KUKA KRL program: MyProgram_046().src

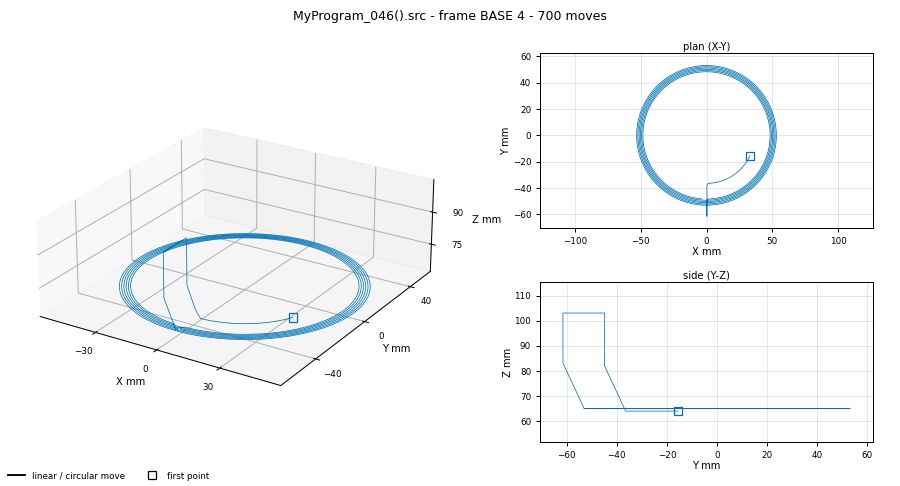
[picture p0: tool path of MyProgram_046().src in frame BASE 4, 700 of 700 moves have a stored position in this frame; points joined in program order, loops and branches not executed]
&ACCESS RVP
&REL 1
&PARAM TEMPLATE = C:\KRC\Roboter\Template\vorgabe
&PARAM EDITMASK = *
DEF MyProgram_046()
; ---- Setting reference (Base) ----
$BASE = BASE_DATA[4]

; --------------------------
; ---- Setting tool (TCP) ----
$TOOL = TOOL_DATA[3]
; --------------------------

$VEL.CP = VEL_APROX_PRINT
Startdeposition()
$VEL.CP = VEL_PRINT
LIN {X 32.9822,Y -15.5864,Z 64,A -32.7373,B 24.8477,C -2.8475,E1 25.1437,E2 -244.1821} C_DIS
LIN {X 32.179,Y -17.1845,Z 64,A -35.4809,B 24.8484,C -2.8403,E1 25.1402,E2 -241.4362} C_DIS
LIN {X 31.292,Y -18.7512,Z 64,A -38.3533,B 24.8494,C -2.8317,E1 25.1362,E2 -238.5581} C_DIS
LIN {X 30.3289,Y -20.2722,Z 64,A -41.1594,B 24.8502,C -2.8242,E1 25.1319,E2 -235.7483} C_DIS
LIN {X 29.3067,Y -21.7235,Z 64,A -44.1232,B 24.8512,C -2.8142,E1 25.127,E2 -232.7751} C_DIS
LIN {X 27.9176,Y -23.4819,Z 64,A -47.6149,B 24.8521,C -2.8055,E1 25.1208,E2 -229.2792} C_DIS
LIN {X 26.4275,Y -25.1472,Z 64,A -51.129,B 24.8531,C -2.7969,E1 25.1142,E2 -225.76} C_DIS
LIN {X 24.8238,Y -26.7316,Z 64,A -54.6334,B 24.8539,C -2.7891,E1 25.1071,E2 -222.2517} C_DIS
LIN {X 23.1454,Y -28.1974,Z 64,A -58.1204,B 24.8547,C -2.7816,E1 25.0997,E2 -218.7605} C_DIS
LIN {X 21.3705,Y -29.5653,Z 64,A -61.4314,B 24.8551,C -2.7774,E1 25.0923,E2 -215.4513} C_DIS
LIN {X 19.9064,Y -30.57,Z 64,A -64.2082,B 24.8557,C -2.7722,E1 25.0858,E2 -212.6714} C_DIS
LIN {X 17.934,Y -31.767,Z 64,A -67.344,B 24.8557,C -2.7725,E1 25.0783,E2 -209.5461} C_DIS
LIN {X 16.1118,Y -32.7286,Z 64,A -71.1277,B 24.857,C -2.7596,E1 25.0689,E2 -205.7422} C_DIS
LIN {X 14.241,Y -33.5852,Z 64,A -74.4803,B 24.8576,C -2.7532,E1 25.0603,E2 -202.3826} C_DIS
LIN {X 12.2935,Y -34.3456,Z 64,A -77.5119,B 24.8577,C -2.7523,E1 25.0524,E2 -199.3554} C_DIS
LIN {X 10.5964,Y -34.9065,Z 64,A -80.3398,B 24.8581,C -2.7487,E1 25.0448,E2 -196.5242} C_DIS
LIN {X 8.8621,Y -35.387,Z 64,A -83.152,B 24.8584,C -2.746,E1 25.0372,E2 -193.71} C_DIS
LIN {X 7.1184,Y -35.7786,Z 64,A -86.157,B 24.8589,C -2.741,E1 25.029,E2 -190.6968} C_DIS
LIN {X 4.917,Y -36.1471,Z 64,A -89.4787,B 24.8589,C -2.741,E1 25.0199,E2 -187.3781} C_DIS
LIN {X 3.1411,Y -36.3441,Z 64,A -92.2456,B 24.859,C -2.7399,E1 25.0122,E2 -184.6106} C_DIS
LIN {X 1.2285,Y -36.4591,Z 64,A -95.4915,B 24.8594,C -2.7358,E1 25.0031,E2 -181.356} C_DIS
LIN {X 1.2285,Y -36.4591,Z 64,A -95.4915,B 24.8594,C -2.7358,E1 25.0031,E2 -181.356} C_DIS
Enddeposition()
LIN {X 0.2612,Y -38.5893,Z 68.5315,A -95.5236,B 24.858,C -2.7494,E1 25.0031,E2 -181.356} C_DIS
LIN {X 0.3711,Y -44.9276,Z 82.1262,A -95.4901,B 24.8595,C -2.7353,E1 25.0031,E2 -181.356} C_DIS
LIN {X 0.3711,Y -44.9276,Z 103.1262,A -95.8409,B 24.8439,C -2.8827,E1 25.0031,E2 -181.356} C_DIS
LIN {X 0.2647,Y -61.4887,Z 103.1262,A -96.1468,B 24.8737,C -2.5936,E1 25.0003,E2 -180.3627} C_DIS
LIN {X 0.2647,Y -61.4887,Z 83.1262,A -95.8133,B 24.887,C -2.4533,E1 25.0003,E2 -180.3627} C_DIS
LIN {X 0.2647,Y -55.1494,Z 69.5315,A -95.8444,B 24.8858,C -2.4664,E1 25.0003,E2 -180.3627} C_DIS
LIN {X 0.2647,Y -53.0363,Z 65,A -95.8563,B 24.8854,C -2.4714,E1 25.0003,E2 -180.3627} C_DIS
Startdeposition()
$VEL.CP = VEL_PRINT
LIN {X -1.9523,Y -53.0044,Z 65,A -98.6503,B 24.8861,C -2.4637,E1 24.9925,E2 -177.5499} C_DIS
LIN {X -4.5507,Y -52.8447,Z 65,A -101.4628,B 24.8861,C -2.4637,E1 24.9846,E2 -174.7363} C_DIS
LIN {X -7.1382,Y -52.5578,Z 65,A -104.2762,B 24.8861,C -2.4641,E1 24.9768,E2 -171.9219} C_DIS
LIN {X -9.7085,Y -52.1442,Z 65,A -107.0908,B 24.886,C -2.4649,E1 24.9691,E2 -169.1066} C_DIS
LIN {X -12.2554,Y -51.605,Z 65,A -109.9063,B 24.8858,C -2.4662,E1 24.9614,E2 -166.2905} C_DIS
LIN {X -14.7728,Y -50.9415,Z 65,A -112.7228,B 24.8857,C -2.4679,E1 24.9538,E2 -163.4736} C_DIS
LIN {X -17.2546,Y -50.1553,Z 65,A -115.5402,B 24.8855,C -2.4699,E1 24.9464,E2 -160.6559} C_DIS
LIN {X -19.6948,Y -49.2482,Z 65,A -118.3587,B 24.8853,C -2.4724,E1 24.939,E2 -157.8374} C_DIS
LIN {X -22.0875,Y -48.2225,Z 65,A -121.178,B 24.885,C -2.4753,E1 24.9318,E2 -155.0181} C_DIS
LIN {X -24.4271,Y -47.0807,Z 65,A -123.9982,B 24.8847,C -2.4786,E1 24.9248,E2 -152.1982} C_DIS
LIN {X -26.7078,Y -45.8254,Z 65,A -126.8195,B 24.8844,C -2.4822,E1 24.9179,E2 -149.3774} C_DIS
LIN {X -28.9242,Y -44.4597,Z 65,A -129.6416,B 24.884,C -2.4863,E1 24.9113,E2 -146.5559} C_DIS
LIN {X -31.0709,Y -42.9869,Z 65,A -132.4651,B 24.8836,C -2.4906,E1 24.9048,E2 -143.7331} C_DIS
LIN {X -33.1427,Y -41.4105,Z 65,A -135.2883,B 24.8831,C -2.4954,E1 24.8986,E2 -140.911} C_DIS
LIN {X -35.1347,Y -39.7344,Z 65,A -138.1128,B 24.8826,C -2.5005,E1 24.8926,E2 -138.0876} C_DIS
LIN {X -37.0421,Y -37.9626,Z 65,A -140.9383,B 24.8821,C -2.5059,E1 24.8869,E2 -135.2634} C_DIS
LIN {X -38.8602,Y -36.0993,Z 65,A -143.7646,B 24.8816,C -2.5117,E1 24.8815,E2 -132.4386} C_DIS
LIN {X -40.5847,Y -34.149,Z 65,A -146.5914,B 24.881,C -2.5178,E1 24.8763,E2 -129.6134} C_DIS
LIN {X -42.1707,Y -32.1693,Z 65,A -149.3664,B 24.8804,C -2.5236,E1 24.8716,E2 -126.8393} C_DIS
LIN {X -43.7019,Y -30.0563,Z 65,A -152.1992,B 24.8798,C -2.5303,E1 24.867,E2 -124.0085} C_DIS
LIN {X -45.1561,Y -27.8244,Z 65,A -155.076,B 24.8791,C -2.5376,E1 24.8627,E2 -121.1346} C_DIS
LIN {X -46.467,Y -25.5752,Z 65,A -157.9055,B 24.8784,C -2.5447,E1 24.8588,E2 -118.3073} C_DIS
LIN {X -47.666,Y -23.2643,Z 65,A -160.7354,B 24.8777,C -2.5521,E1 24.8553,E2 -115.4798} C_DIS
LIN {X -48.7501,Y -20.8975,Z 65,A -163.5659,B 24.877,C -2.5596,E1 24.852,E2 -112.6518} C_DIS
LIN {X -49.7167,Y -18.4802,Z 65,A -166.3969,B 24.8763,C -2.5674,E1 24.8492,E2 -109.8234} C_DIS
LIN {X -50.5636,Y -16.0185,Z 65,A -169.2282,B 24.8755,C -2.5753,E1 24.8467,E2 -106.9949} C_DIS
LIN {X -51.2887,Y -13.5182,Z 65,A -172.0599,B 24.8747,C -2.5834,E1 24.8446,E2 -104.1661} C_DIS
LIN {X -51.8902,Y -10.9852,Z 65,A -174.8919,B 24.8739,C -2.5916,E1 24.8429,E2 -101.337} C_DIS
LIN {X -52.3668,Y -8.4259,Z 65,A -177.7242,B 24.8731,C -2.5999,E1 24.8415,E2 -98.5077} C_DIS
LIN {X -52.7171,Y -5.8462,Z 65,A 179.4433,B 24.8723,C -2.6083,E1 24.8406,E2 -95.6784} C_DIS
LIN {X -52.9405,Y -3.2525,Z 65,A 176.6107,B 24.8714,C -2.6167,E1 24.84,E2 -92.8491} C_DIS
LIN {X -53.0363,Y -0.6509,Z 65,A 173.778,B 24.8706,C -2.6253,E1 24.8398,E2 -90.0197} C_DIS
LIN {X -53.0044,Y 1.9523,Z 65,A 170.9453,B 24.8697,C -2.6338,E1 24.84,E2 -87.1903} C_DIS
LIN {X -52.8447,Y 4.5507,Z 65,A 168.1125,B 24.8689,C -2.6424,E1 24.8405,E2 -84.3609} C_DIS
LIN {X -52.5578,Y 7.1382,Z 65,A 165.2797,B 24.868,C -2.6509,E1 24.8415,E2 -81.5316} C_DIS
LIN {X -52.1442,Y 9.7085,Z 65,A 162.4469,B 24.8672,C -2.6594,E1 24.8429,E2 -78.7024} C_DIS
LIN {X -51.605,Y 12.2554,Z 65,A 159.6143,B 24.8663,C -2.6679,E1 24.8446,E2 -75.8733} C_DIS
LIN {X -50.9415,Y 14.7728,Z 65,A 156.7819,B 24.8655,C -2.6762,E1 24.8467,E2 -73.0445} C_DIS
LIN {X -50.1553,Y 17.2546,Z 65,A 153.9497,B 24.8647,C -2.6845,E1 24.8492,E2 -70.2159} C_DIS
LIN {X -49.2482,Y 19.6948,Z 65,A 151.1178,B 24.8638,C -2.6927,E1 24.852,E2 -67.3875} C_DIS
LIN {X -48.2225,Y 22.0875,Z 65,A 148.2862,B 24.863,C -2.7007,E1 24.8552,E2 -64.5595} C_DIS
LIN {X -47.0807,Y 24.4271,Z 65,A 145.455,B 24.8622,C -2.7085,E1 24.8588,E2 -61.732} C_DIS
LIN {X -45.8254,Y 26.7078,Z 65,A 142.6243,B 24.8614,C -2.7162,E1 24.8626,E2 -58.9048} C_DIS
LIN {X -44.4597,Y 28.9242,Z 65,A 139.7938,B 24.8607,C -2.7237,E1 24.8669,E2 -56.0779} C_DIS
LIN {X -42.9869,Y 31.0709,Z 65,A 136.9641,B 24.8599,C -2.731,E1 24.8714,E2 -53.2516} C_DIS
LIN {X -41.4105,Y 33.1427,Z 65,A 134.1348,B 24.8592,C -2.738,E1 24.8763,E2 -50.4258} C_DIS
LIN {X -39.7344,Y 35.1347,Z 65,A 131.3062,B 24.8585,C -2.7449,E1 24.8814,E2 -47.6007} C_DIS
LIN {X -37.9626,Y 37.0421,Z 65,A 128.4781,B 24.8578,C -2.7514,E1 24.8868,E2 -44.7759} C_DIS
LIN {X -36.0993,Y 38.8602,Z 65,A 125.6675,B 24.8571,C -2.7579,E1 24.8925,E2 -41.9693} C_DIS
LIN {X -34.149,Y 40.5847,Z 65,A 122.8241,B 24.8565,C -2.7636,E1 24.8985,E2 -39.1283} C_DIS
LIN {X -32.1165,Y 42.2114,Z 65,A 119.998,B 24.856,C -2.7693,E1 24.9047,E2 -36.3054} C_DIS
LIN {X -30.0066,Y 43.7365,Z 65,A 117.1728,B 24.8554,C -2.7746,E1 24.9112,E2 -33.4832} C_DIS
LIN {X -27.8244,Y 45.1561,Z 65,A 114.3485,B 24.8549,C -2.7796,E1 24.9178,E2 -30.6618} C_DIS
LIN {X -25.5752,Y 46.467,Z 65,A 111.5249,B 24.8544,C -2.7842,E1 24.9247,E2 -27.841} C_DIS
LIN {X -23.2643,Y 47.666,Z 65,A 108.7023,B 24.8539,C -2.7885,E1 24.9317,E2 -25.0211} C_DIS
LIN {X -20.8975,Y 48.7501,Z 65,A 105.8804,B 24.8535,C -2.7925,E1 24.9389,E2 -22.2018} C_DIS
LIN {X -18.4802,Y 49.7167,Z 65,A 103.0594,B 24.8531,C -2.796,E1 24.9462,E2 -19.3833} C_DIS
LIN {X -16.0185,Y 50.5636,Z 65,A 100.2394,B 24.8528,C -2.7992,E1 24.9537,E2 -16.5656} C_DIS
LIN {X -13.5182,Y 51.2887,Z 65,A 97.4203,B 24.8525,C -2.8019,E1 24.9613,E2 -13.7487} C_DIS
LIN {X -10.9852,Y 51.8902,Z 65,A 94.6021,B 24.8523,C -2.8043,E1 24.969,E2 -10.9325} C_DIS
LIN {X -8.4259,Y 52.3668,Z 65,A 91.7849,B 24.8521,C -2.8063,E1 24.9767,E2 -8.1172} C_DIS
LIN {X -5.8462,Y 52.7171,Z 65,A 88.9687,B 24.8519,C -2.8078,E1 24.9845,E2 -5.3028} C_DIS
LIN {X -3.2525,Y 52.9405,Z 65,A 86.1535,B 24.8518,C -2.809,E1 24.9923,E2 -2.4892} C_DIS
LIN {X -0.6509,Y 53.0363,Z 65,A 83.3685,B 24.8516,C -2.8102,E1 25.0001,E2 0.2932} C_DIS
LIN {X 1.9523,Y 53.0044,Z 65,A 80.5261,B 24.8516,C -2.81,E1 25.0081,E2 3.1355} C_DIS
LIN {X 4.5507,Y 52.8447,Z 65,A 77.7139,B 24.8516,C -2.81,E1 25.0159,E2 5.9466} C_DIS
LIN {X 7.1382,Y 52.5578,Z 65,A 74.9027,B 24.8517,C -2.8094,E1 25.0237,E2 8.7569} C_DIS
LIN {X 9.7085,Y 52.1442,Z 65,A 72.0924,B 24.8518,C -2.8085,E1 25.0314,E2 11.5665} C_DIS
LIN {X 12.2554,Y 51.605,Z 65,A 69.283,B 24.852,C -2.8071,E1 25.0391,E2 14.3753} C_DIS
LIN {X 14.7264,Y 50.9546,Z 65,A 66.5128,B 24.8522,C -2.8052,E1 25.0465,E2 17.1456} C_DIS
LIN {X 17.2546,Y 50.1553,Z 65,A 63.6673,B 24.8524,C -2.8032,E1 25.0541,E2 19.9903} C_DIS
LIN {X 19.6948,Y 49.2482,Z 65,A 60.8608,B 24.8527,C -2.8007,E1 25.0614,E2 22.7967} C_DIS
LIN {X 22.0875,Y 48.2225,Z 65,A 58.0553,B 24.853,C -2.7977,E1 25.0685,E2 25.6023} C_DIS
LIN {X 24.4271,Y 47.0807,Z 65,A 55.2508,B 24.8533,C -2.7944,E1 25.0755,E2 28.4071} C_DIS
LIN {X 26.7078,Y 45.8254,Z 65,A 52.4472,B 24.8537,C -2.7907,E1 25.0823,E2 31.2112} C_DIS
LIN {X 28.9242,Y 44.4597,Z 65,A 49.6444,B 24.8541,C -2.7866,E1 25.089,E2 34.0147} C_DIS
LIN {X 31.0709,Y 42.9869,Z 65,A 46.8424,B 24.8546,C -2.7822,E1 25.0954,E2 36.8175} C_DIS
LIN {X 33.1427,Y 41.4105,Z 65,A 44.0412,B 24.8551,C -2.7774,E1 25.1015,E2 39.6197} C_DIS
LIN {X 35.1347,Y 39.7344,Z 65,A 41.2409,B 24.8556,C -2.7723,E1 25.1074,E2 42.4211} C_DIS
LIN {X 37.0421,Y 37.9626,Z 65,A 38.4413,B 24.8562,C -2.7668,E1 25.1131,E2 45.222} C_DIS
LIN {X 38.796,Y 36.1675,Z 65,A 35.714,B 24.8568,C -2.7607,E1 25.1184,E2 47.952} C_DIS
LIN {X 40.5847,Y 34.149,Z 65,A 32.8444,B 24.8574,C -2.7551,E1 25.1236,E2 50.8221} C_DIS
LIN {X 42.2114,Y 32.1165,Z 65,A 30.0469,B 24.8581,C -2.7487,E1 25.1284,E2 53.6213} C_DIS
LIN {X 43.7365,Y 30.0066,Z 65,A 27.2501,B 24.8588,C -2.7422,E1 25.1329,E2 56.4201} C_DIS
LIN {X 45.1561,Y 27.8244,Z 65,A 24.4538,B 24.8595,C -2.7353,E1 25.1371,E2 59.2185} C_DIS
LIN {X 46.467,Y 25.5752,Z 65,A 21.6582,B 24.8602,C -2.7283,E1 25.141,E2 62.0162} C_DIS
LIN {X 47.666,Y 23.2643,Z 65,A 18.863,B 24.861,C -2.721,E1 25.1445,E2 64.8138} C_DIS
LIN {X 48.7501,Y 20.8975,Z 65,A 16.0683,B 24.8617,C -2.7135,E1 25.1476,E2 67.611} C_DIS
LIN {X 49.7167,Y 18.4802,Z 65,A 13.2739,B 24.8625,C -2.7058,E1 25.1505,E2 70.408} C_DIS
LIN {X 50.5636,Y 16.0185,Z 65,A 10.4801,B 24.8633,C -2.698,E1 25.1529,E2 73.2046} C_DIS
LIN {X 51.2887,Y 13.5181,Z 65,A 7.6866,B 24.8641,C -2.69,E1 25.155,E2 76.0009} C_DIS
LIN {X 51.8902,Y 10.9852,Z 65,A 4.8934,B 24.8649,C -2.6819,E1 25.1567,E2 78.797} C_DIS
LIN {X 52.3668,Y 8.4259,Z 65,A 2.1003,B 24.8658,C -2.6737,E1 25.158,E2 81.5932} C_DIS
LIN {X 52.7171,Y 5.8462,Z 65,A -0.6924,B 24.8666,C -2.6654,E1 25.159,E2 84.3891} C_DIS
LIN {X 52.9268,Y 3.4546,Z 65,A -3.2676,B 24.8674,C -2.6577,E1 25.1596,E2 86.9671} C_DIS
LIN {X 53.033,Y 0.8307,Z 65,A -6.148,B 24.8683,C -2.6479,E1 25.1598,E2 89.8536} C_DIS
LIN {X 53.0044,Y -1.9523,Z 65,A -9.0698,B 24.8691,C -2.6402,E1 25.1596,E2 92.7763} C_DIS
LIN {X 52.8447,Y -4.5507,Z 65,A -11.8622,B 24.87,C -2.6317,E1 25.159,E2 95.5721} C_DIS
LIN {X 52.5578,Y -7.1382,Z 65,A -14.6546,B 24.8708,C -2.6233,E1 25.1581,E2 98.3679} C_DIS
LIN {X 52.1442,Y -9.7085,Z 65,A -17.4472,B 24.8716,C -2.6149,E1 25.1567,E2 101.164} C_DIS
LIN {X 51.605,Y -12.2554,Z 65,A -20.2399,B 24.8724,C -2.6065,E1 25.155,E2 103.9602} C_DIS
LIN {X 50.9415,Y -14.7728,Z 65,A -23.0326,B 24.8733,C -2.5982,E1 25.1529,E2 106.7566} C_DIS
LIN {X 50.1553,Y -17.2546,Z 65,A -25.8256,B 24.8741,C -2.59,E1 25.1505,E2 109.5531} C_DIS
LIN {X 49.2482,Y -19.6948,Z 65,A -28.619,B 24.8748,C -2.5819,E1 25.1477,E2 112.3501} C_DIS
LIN {X 48.2225,Y -22.0875,Z 65,A -31.4126,B 24.8756,C -2.574,E1 25.1445,E2 115.1473} C_DIS
LIN {X 47.0807,Y -24.4271,Z 65,A -34.2065,B 24.8764,C -2.5662,E1 25.141,E2 117.9447} C_DIS
LIN {X 45.8254,Y -26.7078,Z 65,A -37.0009,B 24.8771,C -2.5586,E1 25.1372,E2 120.7427} C_DIS
LIN {X 44.4597,Y -28.9242,Z 65,A -39.7957,B 24.8778,C -2.5511,E1 25.133,E2 123.5411} C_DIS
LIN {X 42.9869,Y -31.0709,Z 65,A -42.5685,B 24.8785,C -2.5443,E1 25.1285,E2 126.3163} C_DIS
LIN {X 41.4105,Y -33.1427,Z 65,A -45.3867,B 24.8792,C -2.5368,E1 25.1237,E2 129.139} C_DIS
LIN {X 39.7344,Y -35.1347,Z 65,A -48.183,B 24.8798,C -2.53,E1 25.1186,E2 131.9387} C_DIS
LIN {X 37.9626,Y -37.0421,Z 65,A -50.98,B 24.8805,C -2.5235,E1 25.1132,E2 134.739} C_DIS
LIN {X 36.0993,Y -38.8602,Z 65,A -53.7777,B 24.8811,C -2.5172,E1 25.1075,E2 137.54} C_DIS
LIN {X 34.149,Y -40.5847,Z 65,A -56.5759,B 24.8816,C -2.5112,E1 25.1016,E2 140.3414} C_DIS
LIN {X 32.1165,Y -42.2114,Z 65,A -59.3749,B 24.8822,C -2.5056,E1 25.0954,E2 143.1435} C_DIS
LIN {X 30.0066,Y -43.7365,Z 65,A -62.1745,B 24.8827,C -2.5002,E1 25.089,E2 145.9462} C_DIS
LIN {X 27.8244,Y -45.1561,Z 65,A -64.9751,B 24.8831,C -2.4952,E1 25.0824,E2 148.7497} C_DIS
LIN {X 25.5752,Y -46.467,Z 65,A -67.7765,B 24.8836,C -2.4904,E1 25.0756,E2 151.5539} C_DIS
LIN {X 23.2643,Y -47.666,Z 65,A -70.5786,B 24.884,C -2.4861,E1 25.0686,E2 154.3586} C_DIS
LIN {X 20.8975,Y -48.7501,Z 65,A -73.3816,B 24.8844,C -2.4821,E1 25.0615,E2 157.1643} C_DIS
LIN {X 18.4802,Y -49.7167,Z 65,A -76.1855,B 24.8847,C -2.4785,E1 25.0542,E2 159.9707} C_DIS
LIN {X 16.0185,Y -50.5636,Z 65,A -78.9903,B 24.885,C -2.4752,E1 25.0467,E2 162.7778} C_DIS
LIN {X 13.5182,Y -51.2887,Z 65,A -81.796,B 24.8853,C -2.4724,E1 25.0392,E2 165.5857} C_DIS
LIN {X 10.9852,Y -51.8902,Z 65,A -84.6027,B 24.8855,C -2.4699,E1 25.0315,E2 168.3945} C_DIS
LIN {X 8.4259,Y -52.3668,Z 65,A -87.4103,B 24.8857,C -2.4678,E1 25.0238,E2 171.204} C_DIS
LIN {X 5.8462,Y -52.7171,Z 65,A -90.2189,B 24.8858,C -2.4662,E1 25.016,E2 174.0143} C_DIS
LIN {X 3.2525,Y -52.9405,Z 65,A -93.0284,B 24.886,C -2.4649,E1 25.0082,E2 176.8254} C_DIS
LIN {X 0.6509,Y -53.0363,Z 65,A -95.8388,B 24.886,C -2.4641,E1 25.0003,E2 179.6373} C_DIS
LIN {X 0.6509,Y -53.0363,Z 65,A -95.8388,B 24.886,C -2.4641,E1 25.0003,E2 179.6373} C_DIS
Enddeposition()
LIN {X 0.2674,Y -52.094,Z 65,A -96.0501,B 24.8842,C -2.4843,E1 24.9999,E2 179.8006} C_DIS
Startdeposition()
$VEL.CP = VEL_PRINT
LIN {X 2.0163,Y -52.0583,Z 65,A -93.0029,B 24.8822,C -2.5055,E1 25.0085,E2 176.7036} C_DIS
LIN {X 3.6967,Y -51.9658,Z 65,A -90.8109,B 24.8815,C -2.5127,E1 25.0147,E2 174.4955} C_DIS
LIN {X 6.9833,Y -51.6275,Z 65,A -87.554,B 24.882,C -2.5077,E1 25.0236,E2 171.2528} C_DIS
LIN {X 9.5679,Y -51.2115,Z 65,A -84.7055,B 24.8818,C -2.5094,E1 25.0315,E2 168.4035} C_DIS
LIN {X 12.0624,Y -50.682,Z 65,A -81.8008,B 24.8814,C -2.5138,E1 25.0394,E2 165.4921} C_DIS
LIN {X 13.8796,Y -50.2148,Z 65,A -79.5679,B 24.8809,C -2.5193,E1 25.0455,E2 163.2498} C_DIS
LIN {X 16.8637,Y -49.2925,Z 65,A -76.8121,B 24.8817,C -2.5102,E1 25.0527,E2 160.5208} C_DIS
LIN {X 20.1169,Y -48.0563,Z 65,A -72.5916,B 24.8805,C -2.523,E1 25.0638,E2 156.2792} C_DIS
LIN {X 22.5196,Y -46.9782,Z 65,A -69.6995,B 24.8801,C -2.5274,E1 25.0711,E2 153.384} C_DIS
LIN {X 24.7919,Y -45.8197,Z 65,A -66.4913,B 24.8789,C -2.5401,E1 25.079,E2 150.1547} C_DIS
LIN {X 27.5966,Y -44.1872,Z 65,A -63.2625,B 24.8789,C -2.5398,E1 25.0867,E2 146.9368} C_DIS
LIN {X 29.763,Y -42.758,Z 65,A -60.4518,B 24.8785,C -2.5445,E1 25.0932,E2 144.1245} C_DIS
LIN {X 31.7714,Y -41.2875,Z 65,A -57.7368,B 24.878,C -2.5497,E1 25.0993,E2 141.407} C_DIS
LIN {X 33.6832,Y -39.7434,Z 65,A -55.1608,B 24.8776,C -2.553,E1 25.1048,E2 138.8329} C_DIS
LIN {X 35.444,Y -38.1818,Z 65,A -52.3705,B 24.8767,C -2.563,E1 25.1106,E2 136.0301} C_DIS
LIN {X 37.5054,Y -36.1583,Z 65,A -49.3954,B 24.8763,C -2.5665,E1 25.1165,E2 133.0595} C_DIS
LIN {X 39.2044,Y -34.3088,Z 65,A -46.6769,B 24.8758,C -2.5725,E1 25.1215,E2 130.3389} C_DIS
LIN {X 40.665,Y -32.5658,Z 65,A -44.1329,B 24.8751,C -2.5798,E1 25.126,E2 127.7893} C_DIS
LIN {X 42.2177,Y -30.5259,Z 65,A -40.472,B 24.8726,C -2.6051,E1 25.1321,E2 124.0863} C_DIS
LIN {X 44.5336,Y -27.034,Z 65,A -36.6989,B 24.8731,C -2.6002,E1 25.1377,E2 120.3438} C_DIS
LIN {X 45.8183,Y -24.7944,Z 65,A -33.875,B 24.8723,C -2.6079,E1 25.1416,E2 117.5162} C_DIS
LIN {X 47.1338,Y -22.1932,Z 65,A -29.8761,B 24.8697,C -2.6343,E1 25.1465,E2 113.4766} C_DIS
LIN {X 48.7949,Y -18.2534,Z 65,A -26.3054,B 24.8707,C -2.6242,E1 25.1501,E2 109.9494} C_DIS
LIN {X 49.5629,Y -16.0498,Z 65,A -23.4351,B 24.8693,C -2.6385,E1 25.1527,E2 107.0616} C_DIS
LIN {X 50.2962,Y -13.5785,Z 65,A -20.6282,B 24.8685,C -2.6467,E1 25.1548,E2 104.2515} C_DIS
LIN {X 50.9451,Y -10.896,Z 65,A -17.6314,B 24.8676,C -2.6553,E1 25.1567,E2 101.2515} C_DIS
LIN {X 51.4547,Y -8.1566,Z 65,A -14.6003,B 24.8667,C -2.6642,E1 25.1581,E2 98.2172} C_DIS
LIN {X 51.8038,Y -5.5188,Z 65,A -11.8131,B 24.8661,C -2.6704,E1 25.1591,E2 95.4317} C_DIS
LIN {X 52.0272,Y -2.6982,Z 65,A -8.3964,B 24.8644,C -2.6868,E1 25.1597,E2 91.9967} C_DIS
LIN {X 52.0967,Y -0.1503,Z 65,A -5.794,B 24.864,C -2.6913,E1 25.1597,E2 89.3991} C_DIS
LIN {X 52.0312,Y 2.6266,Z 65,A -2.9509,B 24.8635,C -2.6964,E1 25.1595,E2 86.5609} C_DIS
LIN {X 51.8478,Y 5.0968,Z 65,A -0.1126,B 24.8624,C -2.7073,E1 25.1588,E2 83.7136} C_DIS
LIN {X 51.5495,Y 7.5347,Z 65,A 2.6369,B 24.8614,C -2.7167,E1 25.1578,E2 80.9581} C_DIS
LIN {X 51.1043,Y 10.1248,Z 65,A 5.5374,B 24.8605,C -2.7257,E1 25.1563,E2 78.0532} C_DIS
LIN {X 50.5209,Y 12.7192,Z 65,A 8.4592,B 24.8596,C -2.7344,E1 25.1544,E2 75.1277} C_DIS
LIN {X 49.7677,Y 15.4031,Z 65,A 11.3708,B 24.859,C -2.7403,E1 25.1521,E2 72.2189} C_DIS
LIN {X 48.9905,Y 17.7209,Z 65,A 14.0882,B 24.8581,C -2.7487,E1 25.1496,E2 69.4969} C_DIS
LIN {X 48.298,Y 19.5293,Z 65,A 16.2864,B 24.8573,C -2.7562,E1 25.1473,E2 67.2931} C_DIS
LIN {X 47.2341,Y 21.9777,Z 65,A 18.9942,B 24.857,C -2.7596,E1 25.1442,E2 64.592} C_DIS
LIN {X 46.0699,Y 24.3238,Z 65,A 22.4058,B 24.855,C -2.7784,E1 25.1398,E2 61.1539} C_DIS
LIN {X 44.8451,Y 26.5141,Z 65,A 25.059,B 24.8545,C -2.7834,E1 25.1361,E2 58.5025} C_DIS
LIN {X 43.0254,Y 29.3758,Z 65,A 28.4002,B 24.8543,C -2.7848,E1 25.131,E2 55.1749} C_DIS
LIN {X 41.527,Y 31.4583,Z 65,A 31.1995,B 24.8537,C -2.7911,E1 25.1263,E2 52.374} C_DIS
LIN {X 39.9445,Y 33.4448,Z 65,A 34.085,B 24.8528,C -2.7994,E1 25.1212,E2 49.4821} C_DIS
LIN {X 38.0022,Y 35.6359,Z 65,A 37.1845,B 24.8523,C -2.804,E1 25.1154,E2 46.3854} C_DIS
LIN {X 36.2083,Y 37.4573,Z 65,A 39.8416,B 24.852,C -2.8067,E1 25.1101,E2 43.733} C_DIS
LIN {X 34.0914,Y 39.3943,Z 65,A 43.1468,B 24.851,C -2.8159,E1 25.1032,E2 40.4195} C_DIS
LIN {X 32.0702,Y 41.0569,Z 65,A 45.9906,B 24.8506,C -2.8204,E1 25.097,E2 37.5756} C_DIS
LIN {X 30.0914,Y 42.528,Z 65,A 48.5016,B 24.8505,C -2.821,E1 25.0914,E2 35.072} C_DIS
LIN {X 28.0762,Y 43.8841,Z 65,A 51.4572,B 24.8495,C -2.8308,E1 25.0845,E2 32.103} C_DIS
LIN {X 25.5344,Y 45.4103,Z 65,A 54.7412,B 24.8489,C -2.8358,E1 25.0765,E2 28.8171} C_DIS
LIN {X 23.1295,Y 46.6809,Z 65,A 57.682,B 24.8486,C -2.8386,E1 25.0692,E2 25.8777} C_DIS
LIN {X 20.6075,Y 47.8483,Z 65,A 60.7564,B 24.8482,C -2.8423,E1 25.0614,E2 22.8021} C_DIS
LIN {X 17.9745,Y 48.898,Z 65,A 63.8199,B 24.848,C -2.8442,E1 25.0534,E2 19.7408} C_DIS
LIN {X 15.4367,Y 49.7573,Z 65,A 66.3532,B 24.8486,C -2.8388,E1 25.0467,E2 17.225} C_DIS
LIN {X 13.6569,Y 50.275,Z 65,A 68.7524,B 24.8477,C -2.8468,E1 25.0402,E2 14.8107} C_DIS
LIN {X 11.2503,Y 50.8678,Z 65,A 71.5362,B 24.8475,C -2.8493,E1 25.0327,E2 12.0249} C_DIS
LIN {X 8.7709,Y 51.3535,Z 65,A 74.2879,B 24.8475,C -2.8499,E1 25.0251,E2 9.275} C_DIS
LIN {X 6.3341,Y 51.7111,Z 65,A 76.9981,B 24.8473,C -2.8505,E1 25.0176,E2 6.5655} C_DIS
LIN {X 3.7754,Y 51.9605,Z 65,A 80.1327,B 24.8467,C -2.8562,E1 25.0088,E2 3.4189} C_DIS
LIN {X 1.1574,Y 52.0843,Z 65,A 82.7925,B 24.8472,C -2.8519,E1 25.0014,E2 0.7699} C_DIS
LIN {X -1.5988,Y 52.0723,Z 65,A 85.5959,B 24.8477,C -2.8472,E1 24.9937,E2 -2.0224} C_DIS
LIN {X -3.7831,Y 51.96,Z 65,A 88.1184,B 24.8476,C -2.8483,E1 24.9866,E2 -4.5483} C_DIS
LIN {X -6.4156,Y 51.701,Z 65,A 90.9182,B 24.848,C -2.8448,E1 24.9789,E2 -7.3416} C_DIS
LIN {X -9.2959,Y 51.2608,Z 65,A 94.2488,B 24.848,C -2.8448,E1 24.9697,E2 -10.6752} C_DIS
LIN {X -11.9018,Y 50.7194,Z 65,A 97.1229,B 24.8483,C -2.8413,E1 24.9619,E2 -13.5446} C_DIS
LIN {X -14.233,Y 50.1149,Z 65,A 99.8698,B 24.8484,C -2.8403,E1 24.9544,E2 -16.2933} C_DIS
LIN {X -17.4327,Y 49.094,Z 65,A 103.9771,B 24.8482,C -2.8428,E1 24.9435,E2 -20.4144} C_DIS
LIN {X -20.724,Y 47.7975,Z 65,A 107.4263,B 24.8495,C -2.8301,E1 24.9347,E2 -23.8411} C_DIS
LIN {X -24.6426,Y 45.9006,Z 65,A 112.0858,B 24.8506,C -2.8205,E1 24.9231,E2 -28.49} C_DIS
LIN {X -26.8103,Y 44.6696,Z 65,A 115.498,B 24.8499,C -2.8265,E1 24.9148,E2 -31.9268} C_DIS
LIN {X -30.0868,Y 42.5312,Z 65,A 119.5759,B 24.8512,C -2.8146,E1 24.9054,E2 -35.9899} C_DIS
LIN {X -32.5559,Y 40.673,Z 65,A 122.7921,B 24.8522,C -2.8046,E1 24.8984,E2 -39.194} C_DIS
LIN {X -33.9983,Y 39.4749,Z 65,A 125.1682,B 24.8522,C -2.805,E1 24.8933,E2 -41.5804} C_DIS
LIN {X -36.7687,Y 36.9077,Z 65,A 129.0316,B 24.8537,C -2.7908,E1 24.8856,E2 -45.426} C_DIS
LIN {X -39.1493,Y 34.3719,Z 65,A 133.3275,B 24.8539,C -2.7887,E1 24.8775,E2 -49.7359} C_DIS
LIN {X -41.0009,Y 32.141,Z 65,A 136.7579,B 24.8544,C -2.7842,E1 24.8715,E2 -53.1717} C_DIS
LIN {X -44.1302,Y 27.6878,Z 65,A 142.1484,B 24.857,C -2.7588,E1 24.8632,E2 -58.5283} C_DIS
LIN {X -45.4504,Y 25.4626,Z 65,A 145.0063,B 24.8579,C -2.751,E1 24.8592,E2 -61.3824} C_DIS
LIN {X -46.6262,Y 23.2397,Z 65,A 148.2036,B 24.858,C -2.7495,E1 24.8552,E2 -64.5932} C_DIS
LIN {X -48.3944,Y 19.2901,Z 65,A 152.1676,B 24.8607,C -2.7235,E1 24.8508,E2 -68.5169} C_DIS
LIN {X -49.1892,Y 17.1612,Z 65,A 155.1884,B 24.8607,C -2.7237,E1 24.848,E2 -71.5552} C_DIS
LIN {X -50.0925,Y 14.3118,Z 65,A 158.398,B 24.8618,C -2.7124,E1 24.8454,E2 -74.7565} C_DIS
LIN {X -51.0165,Y 10.5548,Z 65,A 162.6795,B 24.8631,C -2.6996,E1 24.8427,E2 -79.0325} C_DIS
LIN {X -51.4778,Y 8.0076,Z 65,A 165.5323,B 24.864,C -2.6908,E1 24.8414,E2 -81.881} C_DIS
LIN {X -51.8055,Y 5.5019,Z 65,A 168.2034,B 24.8651,C -2.6804,E1 24.8405,E2 -84.5434} C_DIS
LIN {X -52.01,Y 3.0091,Z 65,A 171.1056,B 24.8657,C -2.674,E1 24.8399,E2 -87.4477} C_DIS
LIN {X -52.0876,Y 0.9777,Z 65,A 173.5053,B 24.8662,C -2.6694,E1 24.8398,E2 -89.8508} C_DIS
LIN {X -52.0462,Y -2.2971,Z 65,A 177.4946,B 24.8667,C -2.6639,E1 24.8401,E2 -93.851} C_DIS
LIN {X -51.7741,Y -5.7961,Z 65,A -179.06,B 24.8686,C -2.6457,E1 24.8411,E2 -97.2736} C_DIS
LIN {X -51.3921,Y -8.5401,Z 65,A -175.6321,B 24.8689,C -2.6421,E1 24.8426,E2 -100.7132} C_DIS
LIN {X -50.7719,Y -11.6745,Z 65,A -172.741,B 24.8709,C -2.6221,E1 24.8442,E2 -103.5734} C_DIS
LIN {X -50.0186,Y -14.5699,Z 65,A -169.2041,B 24.8715,C -2.616,E1 24.8468,E2 -107.1163} C_DIS
LIN {X -49.0931,Y -17.4353,Z 65,A -165.631,B 24.8721,C -2.6103,E1 24.85,E2 -110.6963} C_DIS
LIN {X -47.6281,Y -21.1126,Z 65,A -161.5744,B 24.8737,C -2.5935,E1 24.8544,E2 -114.7352} C_DIS
LIN {X -46.6441,Y -23.2037,Z 65,A -158.9124,B 24.8742,C -2.5884,E1 24.8576,E2 -117.3994} C_DIS
LIN {X -45.7334,Y -24.951,Z 65,A -156.3547,B 24.8742,C -2.5887,E1 24.8611,E2 -119.9713} C_DIS
LIN {X -43.3955,Y -28.8261,Z 65,A -151.7571,B 24.876,C -2.5701,E1 24.8678,E2 -124.5478} C_DIS
LIN {X -42.4097,Y -30.2572,Z 65,A -149.3779,B 24.8757,C -2.5728,E1 24.8717,E2 -126.9452} C_DIS
LIN {X -40.3687,Y -32.9313,Z 65,A -146.2209,B 24.8774,C -2.5556,E1 24.8772,E2 -130.0759} C_DIS
LIN {X -38.8038,Y -34.7613,Z 65,A -143.5855,B 24.878,C -2.5495,E1 24.882,E2 -132.7087} C_DIS
LIN {X -37.5163,Y -36.147,Z 65,A -140.6851,B 24.8771,C -2.5583,E1 24.8877,E2 -135.6426} C_DIS
LIN {X -34.593,Y -38.9544,Z 65,A -136.898,B 24.879,C -2.5386,E1 24.8954,E2 -139.398} C_DIS
LIN {X -32.5731,Y -40.6591,Z 65,A -134.1078,B 24.8797,C -2.5314,E1 24.9014,E2 -142.1816} C_DIS
LIN {X -30.7855,Y -42.0277,Z 65,A -131.6708,B 24.8802,C -2.5265,E1 24.9068,E2 -144.6157} C_DIS
LIN {X -27.5814,Y -44.1967,Z 65,A -127.4498,B 24.8809,C -2.5193,E1 24.9166,E2 -148.8335} C_DIS
LIN {X -26.3006,Y -44.9713,Z 65,A -125.2762,B 24.8802,C -2.5258,E1 24.9219,E2 -151.0293} C_DIS
LIN {X -23.4771,Y -46.5077,Z 65,A -121.956,B 24.881,C -2.5177,E1 24.9301,E2 -154.3392} C_DIS
LIN {X -20.9421,Y -47.7024,Z 65,A -118.9235,B 24.8814,C -2.5135,E1 24.9378,E2 -157.3691} C_DIS
LIN {X -18.4941,Y -48.7037,Z 65,A -116.3205,B 24.8822,C -2.5055,E1 24.9445,E2 -159.9587} C_DIS
LIN {X -16.6033,Y -49.3803,Z 65,A -113.912,B 24.882,C -2.5072,E1 24.9509,E2 -162.3759} C_DIS
LIN {X -14.1619,Y -50.135,Z 65,A -111.049,B 24.8821,C -2.5062,E1 24.9586,E2 -165.2413} C_DIS
LIN {X -11.6527,Y -50.777,Z 65,A -108.1183,B 24.8821,C -2.5062,E1 24.9665,E2 -168.1759} C_DIS
LIN {X -8.9973,Y -51.3145,Z 65,A -105.1337,B 24.8821,C -2.5052,E1 24.9747,E2 -171.1614} C_DIS
LIN {X -6.2497,Y -51.721,Z 65,A -101.8923,B 24.8819,C -2.508,E1 24.9837,E2 -174.4119} C_DIS
LIN {X -3.0681,Y -52.0068,Z 65,A -98.706,B 24.8825,C -2.502,E1 24.9926,E2 -177.5853} C_DIS
LIN {X -0.7966,Y -52.091,Z 65,A -96.0977,B 24.8823,C -2.5043,E1 24.9999,E2 -180.1994} C_DIS
LIN {X -0.7966,Y -52.091,Z 65,A -96.0977,B 24.8823,C -2.5043,E1 24.9999,E2 -180.1994} C_DIS
Enddeposition()
LIN {X 0.2552,Y -51.1523,Z 65,A -95.2234,B 24.8812,C -2.5156,E1 25.0024,E2 -181.1006} C_DIS
Startdeposition()
$VEL.CP = VEL_PRINT
LIN {X -2.5633,Y -51.0907,Z 65,A -99.8847,B 24.8838,C -2.4885,E1 24.9892,E2 -176.3742} C_DIS
LIN {X -6.9954,Y -50.6742,Z 65,A -104.1628,B 24.8826,C -2.5013,E1 24.9774,E2 -172.124} C_DIS
LIN {X -8.8757,Y -50.3788,Z 65,A -106.5871,B 24.883,C -2.4969,E1 24.9707,E2 -169.687} C_DIS
LIN {X -11.4127,Y -49.8651,Z 65,A -109.6,B 24.883,C -2.4963,E1 24.9624,E2 -166.6688} C_DIS
LIN {X -13.9474,Y -49.2162,Z 65,A -112.7895,B 24.8833,C -2.4937,E1 24.9538,E2 -163.4684} C_DIS
LIN {X -18.1443,Y -47.8283,Z 65,A -117.4308,B 24.8824,C -2.5029,E1 24.9416,E2 -158.8399} C_DIS
LIN {X -20.6244,Y -46.8128,Z 65,A -120.4158,B 24.8821,C -2.5062,E1 24.9339,E2 -155.8559} C_DIS
LIN {X -23.0559,Y -45.6645,Z 65,A -124.0486,B 24.8827,C -2.4998,E1 24.9248,E2 -152.1983} C_DIS
LIN {X -26.0663,Y -44.0149,Z 65,A -127.3231,B 24.8813,C -2.5141,E1 24.9169,E2 -148.9483} C_DIS
LIN {X -28.4386,Y -42.5208,Z 65,A -130.347,B 24.8807,C -2.5208,E1 24.9098,E2 -145.9304} C_DIS
LIN {X -30.6034,Y -40.9902,Z 65,A -133.7852,B 24.8809,C -2.5184,E1 24.902,E2 -142.4745} C_DIS
LIN {X -33.6831,Y -38.4996,Z 65,A -138.024,B 24.8799,C -2.5296,E1 24.893,E2 -138.2462} C_DIS
LIN {X -35.5402,Y -36.7921,Z 65,A -140.6243,B 24.879,C -2.5387,E1 24.8877,E2 -135.6569} C_DIS
LIN {X -37.4815,Y -34.8138,Z 65,A -143.9416,B 24.8787,C -2.542,E1 24.8813,E2 -132.3333} C_DIS
LIN {X -39.3223,Y -32.7189,Z 65,A -147.0506,B 24.878,C -2.5493,E1 24.8756,E2 -129.2274} C_DIS
LIN {X -41.401,Y -30.0455,Z 65,A -150.6149,B 24.8768,C -2.5617,E1 24.8696,E2 -125.6757} C_DIS
LIN {X -42.3175,Y -28.7397,Z 65,A -153.1442,B 24.8774,C -2.5552,E1 24.8656,E2 -123.1182} C_DIS
LIN {X -44.7852,Y -24.7208,Z 65,A -157.5345,B 24.8748,C -2.5819,E1 24.8594,E2 -118.7692} C_DIS
LIN {X -45.6861,Y -23.0139,Z 65,A -160.0598,B 24.8748,C -2.5824,E1 24.8562,E2 -116.2315} C_DIS
LIN {X -46.7663,Y -20.7311,Z 65,A -163.5832,B 24.875,C -2.5802,E1 24.8521,E2 -112.6836} C_DIS
LIN {X -48.4305,Y -16.4703,Z 65,A -167.8462,B 24.8724,C -2.6073,E1 24.848,E2 -108.4613} C_DIS
LIN {X -49.256,Y -13.807,Z 65,A -171.639,B 24.8724,C -2.607,E1 24.8449,E2 -104.6458} C_DIS
LIN {X -49.9341,Y -11.1086,Z 65,A -174.6036,B 24.8713,C -2.6185,E1 24.8431,E2 -101.6914} C_DIS
LIN {X -50.5936,Y -7.5581,Z 65,A -178.0994,B 24.8693,C -2.6386,E1 24.8414,E2 -98.223} C_DIS
LIN {X -50.9599,Y -4.4624,Z 65,A 177.3696,B 24.8696,C -2.6349,E1 24.8401,E2 -93.6558} C_DIS
LIN {X -51.1478,Y -0.8264,Z 65,A 173.0951,B 24.8686,C -2.6449,E1 24.8398,E2 -89.3796} C_DIS
LIN {X -51.0829,Y 2.7057,Z 65,A 169.8496,B 24.8664,C -2.6673,E1 24.8401,E2 -86.168} C_DIS
LIN {X -50.8689,Y 5.3974,Z 65,A 166.8767,B 24.8654,C -2.6775,E1 24.8409,E2 -83.2017} C_DIS
LIN {X -50.5256,Y 7.998,Z 65,A 163.6792,B 24.8648,C -2.6831,E1 24.8422,E2 -79.9985} C_DIS
LIN {X -49.8311,Y 11.5595,Z 65,A 159.698,B 24.8634,C -2.6969,E1 24.8445,E2 -76.027} C_DIS
LIN {X -49.1766,Y 14.0862,Z 65,A 156.4548,B 24.8629,C -2.7014,E1 24.8469,E2 -72.7759} C_DIS
LIN {X -47.8856,Y 17.9933,Z 65,A 152.4921,B 24.8606,C -2.7245,E1 24.8505,E2 -68.8458} C_DIS
LIN {X -47.2997,Y 19.482,Z 65,A 150.2406,B 24.8607,C -2.7234,E1 24.8529,E2 -66.579} C_DIS
LIN {X -45.8756,Y 22.6319,Z 65,A 146.7672,B 24.859,C -2.7404,E1 24.857,E2 -63.1273} C_DIS
LIN {X -44.2029,Y 25.748,Z 65,A 142.9148,B 24.8576,C -2.7532,E1 24.8621,E2 -59.2853} C_DIS
LIN {X -42.2738,Y 28.8048,Z 65,A 138.2641,B 24.8574,C -2.7557,E1 24.8692,E2 -54.617} C_DIS
LIN {X -40.824,Y 30.8251,Z 65,A 135.8632,B 24.856,C -2.7686,E1 24.8731,E2 -52.2354} C_DIS
LIN {X -39.4688,Y 32.5416,Z 65,A 132.7853,B 24.8563,C -2.7658,E1 24.8786,E2 -49.1363} C_DIS
LIN {X -36.897,Y 35.4314,Z 65,A 128.4935,B 24.8552,C -2.7769,E1 24.8867,E2 -44.8523} C_DIS
LIN {X -33.9068,Y 38.303,Z 65,A 124.3477,B 24.8533,C -2.7949,E1 24.8951,E2 -40.7326} C_DIS
LIN {X -32.2958,Y 39.6707,Z 65,A 121.4468,B 24.8536,C -2.792,E1 24.9014,E2 -37.8138} C_DIS
LIN {X -29.3487,Y 41.8981,Z 65,A 117.6661,B 24.8521,C -2.8057,E1 24.9099,E2 -34.0525} C_DIS
LIN {X -26.9022,Y 43.5097,Z 65,A 113.7087,B 24.8526,C -2.8015,E1 24.9192,E2 -30.0725} C_DIS
LIN {X -24.1041,Y 45.1204,Z 65,A 110.2185,B 24.8517,C -2.8095,E1 24.9278,E2 -26.5913} C_DIS
LIN {X -20.5303,Y 46.8539,Z 65,A 106.6443,B 24.8496,C -2.8299,E1 24.9367,E2 -23.0567} C_DIS
LIN {X -18.9273,Y 47.5243,Z 65,A 104.4521,B 24.8496,C -2.8286,E1 24.9424,E2 -20.8567} C_DIS
LIN {X -16.6996,Y 48.3513,Z 65,A 101.2372,B 24.8503,C -2.8232,E1 24.9509,E2 -17.6223} C_DIS
LIN {X -13.4657,Y 49.3504,Z 65,A 97.8279,B 24.8492,C -2.8333,E1 24.96,E2 -14.2317} C_DIS
LIN {X -10.4345,Y 50.079,Z 65,A 94.3806,B 24.8488,C -2.8371,E1 24.9694,E2 -10.789} C_DIS
LIN {X -8.0897,Y 50.5104,Z 65,A 91.3834,B 24.8491,C -2.8337,E1 24.9776,E2 -7.7807} C_DIS
LIN {X -4.8426,Y 50.9248,Z 65,A 87.9643,B 24.8485,C -2.8398,E1 24.9871,E2 -4.3739} C_DIS
LIN {X -2.3531,Y 51.1004,Z 65,A 85.1441,B 24.8485,C -2.8404,E1 24.995,E2 -1.5544} C_DIS
LIN {X 1.0131,Y 51.1444,Z 65,A 81.7008,B 24.8477,C -2.8467,E1 25.0045,E2 1.8738} C_DIS
LIN {X 4.4547,Y 50.9606,Z 65,A 77.6639,B 24.8481,C -2.8437,E1 25.0158,E2 5.9163} C_DIS
LIN {X 6.8081,Y 50.6998,Z 65,A 74.9205,B 24.8483,C -2.8416,E1 25.0234,E2 8.6625} C_DIS
LIN {X 9.2683,Y 50.3082,Z 65,A 72.0974,B 24.8485,C -2.8401,E1 25.0312,E2 11.4863} C_DIS
LIN {X 12.7267,Y 49.5459,Z 65,A 67.4686,B 24.8499,C -2.8263,E1 25.0438,E2 16.1413} C_DIS
LIN {X 16.1558,Y 48.5365,Z 65,A 64.0619,B 24.8491,C -2.8339,E1 25.0528,E2 19.5237} C_DIS
LIN {X 18.7543,Y 47.5925,Z 65,A 61,B 24.8494,C -2.8316,E1 25.0608,E2 22.5844} C_DIS
LIN {X 21.4576,Y 46.4366,Z 65,A 57.6724,B 24.8498,C -2.8274,E1 25.0693,E2 25.9138} C_DIS
LIN {X 23.545,Y 45.4146,Z 65,A 55.3405,B 24.8496,C -2.8292,E1 25.0751,E2 28.2352} C_DIS
LIN {X 25.5694,Y 44.3055,Z 65,A 52.5446,B 24.8504,C -2.8217,E1 25.0819,E2 31.0405} C_DIS
LIN {X 27.2966,Y 43.2629,Z 65,A 49.683,B 24.852,C -2.8071,E1 25.0888,E2 33.9276} C_DIS
LIN {X 30.4916,Y 41.0745,Z 65,A 45.9577,B 24.8515,C -2.8114,E1 25.0972,E2 37.6297} C_DIS
LIN {X 32.6378,Y 39.3897,Z 65,A 42.4155,B 24.8531,C -2.7966,E1 25.1049,E2 41.1936} C_DIS
LIN {X 35.5203,Y 36.8113,Z 65,A 38.6594,B 24.8528,C -2.799,E1 25.1125,E2 44.9287} C_DIS
LIN {X 37.4513,Y 34.8458,Z 65,A 34.9435,B 24.8548,C -2.7802,E1 25.1197,E2 48.6729} C_DIS
LIN {X 39.982,Y 31.9103,Z 65,A 31.28,B 24.8545,C -2.7835,E1 25.1262,E2 52.3119} C_DIS
LIN {X 41.5269,Y 29.8718,Z 65,A 28.0834,B 24.8559,C -2.77,E1 25.1315,E2 55.5249} C_DIS
LIN {X 44.0171,Y 26.0626,Z 65,A 23.7039,B 24.8557,C -2.7714,E1 25.1381,E2 59.8792} C_DIS
LIN {X 45.4846,Y 23.408,Z 65,A 19.9512,B 24.8574,C -2.7552,E1 25.1431,E2 63.6506} C_DIS
LIN {X 46.4387,Y 21.4529,Z 65,A 16.6775,B 24.8599,C -2.7317,E1 25.147,E2 66.9621} C_DIS
LIN {X 48.0412,Y 17.573,Z 65,A 12.8842,B 24.8594,C -2.7365,E1 25.1508,E2 70.7229} C_DIS
LIN {X 48.8881,Y 15.0574,Z 65,A 9.3342,B 24.8614,C -2.7161,E1 25.1538,E2 74.301} C_DIS
LIN {X 50.009,Y 10.7652,Z 65,A 4.9809,B 24.8617,C -2.7137,E1 25.1566,E2 78.6349} C_DIS
LIN {X 50.5055,Y 8.1276,Z 65,A 1.9659,B 24.8627,C -2.7043,E1 25.1581,E2 81.6544} C_DIS
LIN {X 50.8508,Y 5.5699,Z 65,A -1.3634,B 24.8645,C -2.6864,E1 25.1592,E2 85.0064} C_DIS
LIN {X 51.1201,Y 1.8942,Z 65,A -4.9094,B 24.8645,C -2.6854,E1 25.1597,E2 88.5337} C_DIS
LIN {X 51.1511,Y -0.6321,Z 65,A -7.4946,B 24.865,C -2.6815,E1 25.1597,E2 91.1126} C_DIS
LIN {X 51.0777,Y -2.7994,Z 65,A -10.2554,B 24.8664,C -2.667,E1 25.1594,E2 93.8912} C_DIS
LIN {X 50.8559,Y -5.5208,Z 65,A -13.3524,B 24.8675,C -2.6566,E1 25.1586,E2 96.9946} C_DIS
LIN {X 50.3699,Y -8.9253,Z 65,A -16.8011,B 24.8679,C -2.6528,E1 25.1571,E2 100.432} C_DIS
LIN {X 49.9288,Y -11.1328,Z 65,A -19.5984,B 24.8692,C -2.6392,E1 25.1555,E2 103.2451} C_DIS
LIN {X 49.2921,Y -13.6795,Z 65,A -22.5523,B 24.8701,C -2.6298,E1 25.1534,E2 106.2042} C_DIS
LIN {X 47.9782,Y -17.7457,Z 65,A -27.2695,B 24.8714,C -2.6167,E1 25.1492,E2 110.926} C_DIS
LIN {X 46.4027,Y -21.5304,Z 65,A -32.4274,B 24.8739,C -2.5915,E1 25.1434,E2 116.1151} C_DIS
LIN {X 44.9719,Y -24.3781,Z 65,A -35.8036,B 24.8745,C -2.5851,E1 25.1389,E2 119.4887} C_DIS
LIN {X 42.9211,Y -27.8317,Z 65,A -39.5866,B 24.8743,C -2.587,E1 25.1334,E2 123.248} C_DIS
LIN {X 41.9504,Y -29.2735,Z 65,A -41.7494,B 24.8753,C -2.5774,E1 25.13,E2 125.4229} C_DIS
LIN {X 40.2875,Y -31.5237,Z 65,A -44.6276,B 24.8756,C -2.5742,E1 25.1252,E2 128.2948} C_DIS
LIN {X 38.8759,Y -33.2482,Z 65,A -47.366,B 24.8767,C -2.563,E1 25.1202,E2 131.0473} C_DIS
LIN {X 37.0737,Y -35.2475,Z 65,A -50.59,B 24.8778,C -2.5514,E1 25.1141,E2 134.2847} C_DIS
LIN {X 35.1176,Y -37.1959,Z 65,A -53.3162,B 24.8778,C -2.5514,E1 25.1086,E2 136.9994} C_DIS
LIN {X 33.3181,Y -38.8163,Z 65,A -55.8627,B 24.8781,C -2.5486,E1 25.1033,E2 139.5425} C_DIS
LIN {X 31.6872,Y -40.1583,Z 65,A -58.4853,B 24.879,C -2.5384,E1 25.0976,E2 142.1793} C_DIS
LIN {X 29.5711,Y -41.7414,Z 65,A -61.3926,B 24.8795,C -2.5334,E1 25.091,E2 145.0881} C_DIS
LIN {X 26.7844,Y -43.582,Z 65,A -65.3151,B 24.8805,C -2.5228,E1 25.0818,E2 149.023} C_DIS
LIN {X 23.7659,Y -45.2985,Z 65,A -68.7196,B 24.8803,C -2.5255,E1 25.0735,E2 152.4113} C_DIS
LIN {X 21.0414,Y -46.6264,Z 65,A -72.7644,B 24.8819,C -2.5078,E1 25.0632,E2 156.4875} C_DIS
LIN {X 18.3444,Y -47.7518,Z 65,A -75.5393,B 24.8815,C -2.5127,E1 25.0561,E2 159.2446} C_DIS
LIN {X 16.2193,Y -48.5151,Z 65,A -79.1891,B 24.8837,C -2.4888,E1 25.0463,E2 162.944} C_DIS
LIN {X 12.2232,Y -49.6726,Z 65,A -82.863,B 24.8825,C -2.5021,E1 25.0365,E2 166.5806} C_DIS
LIN {X 9.7028,Y -50.2257,Z 65,A -85.772,B 24.8828,C -2.4993,E1 25.0285,E2 169.4927} C_DIS
LIN {X 7.0127,Y -50.6717,Z 65,A -89.0267,B 24.8833,C -2.4935,E1 25.0195,E2 172.758} C_DIS
LIN {X 3.4916,Y -51.0351,Z 65,A -92.4958,B 24.8826,C -2.5004,E1 25.0099,E2 176.2087} C_DIS
LIN {X 1.2836,Y -51.139,Z 65,A -95.1765,B 24.8831,C -2.4959,E1 25.0024,E2 178.8994} C_DIS
LIN {X 1.2836,Y -51.139,Z 65,A -95.1765,B 24.8831,C -2.4959,E1 25.0024,E2 178.8994} C_DIS
Enddeposition()
LIN {X 0.2483,Y -50.2075,Z 65,A -95.5643,B 24.8802,C -2.5257,E1 25.0015,E2 179.2163} C_DIS
Startdeposition()
$VEL.CP = VEL_PRINT
LIN {X 2.2629,Y -50.161,Z 65,A -92.8364,B 24.8795,C -2.534,E1 25.0092,E2 176.4693} C_DIS
LIN {X 5.2511,Y -49.9365,Z 65,A -88.9836,B 24.8785,C -2.5436,E1 25.0199,E2 172.596} C_DIS
LIN {X 8.5671,Y -49.4765,Z 65,A -85.4206,B 24.8787,C -2.5416,E1 25.0297,E2 169.0412} C_DIS
LIN {X 11.2453,Y -48.9365,Z 65,A -82.3641,B 24.8786,C -2.5432,E1 25.0381,E2 165.9847} C_DIS
LIN {X 14.7902,Y -47.9843,Z 65,A -77.5399,B 24.877,C -2.5597,E1 25.0511,E2 161.1296} C_DIS
LIN {X 18.0776,Y -46.8451,Z 65,A -74.3675,B 24.878,C -2.5497,E1 25.0593,E2 157.9875} C_DIS
LIN {X 19.7405,Y -46.169,Z 65,A -71.9997,B 24.8771,C -2.5588,E1 25.0655,E2 155.604} C_DIS
LIN {X 22.6756,Y -44.8005,Z 65,A -68.5627,B 24.8771,C -2.5596,E1 25.0741,E2 152.1739} C_DIS
LIN {X 25.0269,Y -43.5303,Z 65,A -65.3301,B 24.8762,C -2.5684,E1 25.082,E2 148.9299} C_DIS
LIN {X 27.3966,Y -42.0802,Z 65,A -61.5627,B 24.8744,C -2.5861,E1 25.0909,E2 145.1328} C_DIS
LIN {X 30.6655,Y -39.76,Z 65,A -57.7223,B 24.8749,C -2.581,E1 25.0995,E2 141.3182} C_DIS
LIN {X 32.0664,Y -38.6391,Z 65,A -55.3319,B 24.8738,C -2.5923,E1 25.1047,E2 138.9103} C_DIS
LIN {X 34.7899,Y -36.2063,Z 65,A -51.8367,B 24.8742,C -2.5885,E1 25.1118,E2 135.4383} C_DIS
LIN {X 35.9209,Y -35.0852,Z 65,A -49.1932,B 24.8722,C -2.6094,E1 25.117,E2 132.7566} C_DIS
LIN {X 38.331,Y -32.4344,Z 65,A -45.6761,B 24.8722,C -2.6081,E1 25.1235,E2 129.2583} C_DIS
LIN {X 40.4557,Y -29.7418,Z 65,A -41.341,B 24.8704,C -2.627,E1 25.1308,E2 124.8992} C_DIS
LIN {X 42.3697,Y -26.9453,Z 65,A -37.8213,B 24.8701,C -2.6305,E1 25.1362,E2 121.3886} C_DIS
LIN {X 43.9116,Y -24.352,Z 65,A -34.6108,B 24.8696,C -2.6356,E1 25.1407,E2 118.1828} C_DIS
LIN {X 45.159,Y -21.9534,Z 65,A -31.3332,B 24.8683,C -2.6485,E1 25.1448,E2 114.8921} C_DIS
LIN {X 46.189,Y -19.6923,Z 65,A -28.4755,B 24.8674,C -2.6574,E1 25.148,E2 112.029} C_DIS
LIN {X 47.5835,Y -16.0324,Z 65,A -23.7635,B 24.8655,C -2.6759,E1 25.1525,E2 107.2995} C_DIS
LIN {X 48.5855,Y -12.6775,Z 65,A -20.1922,B 24.8652,C -2.6795,E1 25.1552,E2 103.7403} C_DIS
LIN {X 49.185,Y -10.1029,Z 65,A -17.4881,B 24.8649,C -2.6825,E1 25.1568,E2 101.0449} C_DIS
LIN {X 49.6918,Y -7.2092,Z 65,A -13.4739,B 24.8624,C -2.7067,E1 25.1586,E2 96.997} C_DIS
LIN {X 50.0459,Y -4.0795,Z 65,A -10.4076,B 24.8624,C -2.7071,E1 25.1594,E2 93.9479} C_DIS
LIN {X 50.1827,Y -1.7191,Z 65,A -7.6533,B 24.8614,C -2.7167,E1 25.1597,E2 91.1871} C_DIS
LIN {X 50.2022,Y 0.9886,Z 65,A -4.1076,B 24.8594,C -2.7359,E1 25.1597,E2 87.6172} C_DIS
LIN {X 49.7988,Y 6.4277,Z 65,A 1.5578,B 24.8586,C -2.7437,E1 25.1582,E2 81.967} C_DIS
LIN {X 49.4122,Y 8.9258,Z 65,A 4.4529,B 24.8577,C -2.7527,E1 25.1569,E2 79.0674} C_DIS
LIN {X 48.8563,Y 11.5892,Z 65,A 7.4816,B 24.8569,C -2.7606,E1 25.155,E2 76.0378} C_DIS
LIN {X 48.3664,Y 13.4895,Z 65,A 9.5022,B 24.8566,C -2.7628,E1 25.1536,E2 74.0236} C_DIS
LIN {X 47.4653,Y 16.3813,Z 65,A 13.2131,B 24.855,C -2.7781,E1 25.1504,E2 70.2976} C_DIS
LIN {X 46.881,Y 17.9847,Z 65,A 15.891,B 24.8529,C -2.7985,E1 25.1476,E2 67.5861} C_DIS
LIN {X 45.3,Y 21.6599,Z 65,A 20.0119,B 24.8525,C -2.8021,E1 25.1428,E2 63.479} C_DIS
LIN {X 43.6439,Y 24.829,Z 65,A 23.6589,B 24.8523,C -2.8043,E1 25.138,E2 59.8461} C_DIS
LIN {X 42.3488,Y 26.9786,Z 65,A 26.4986,B 24.8515,C -2.8111,E1 25.1338,E2 57.0046} C_DIS
LIN {X 40.9031,Y 29.1234,Z 65,A 29.6603,B 24.8503,C -2.8226,E1 25.1288,E2 53.8312} C_DIS
LIN {X 39.4178,Y 31.1042,Z 65,A 32.7423,B 24.8491,C -2.8343,E1 25.1235,E2 50.7359} C_DIS
LIN {X 36.8993,Y 34.0543,Z 65,A 36.7748,B 24.8489,C -2.8364,E1 25.116,E2 46.7166} C_DIS
LIN {X 34.9264,Y 36.0748,Z 65,A 39.3445,B 24.8495,C -2.8305,E1 25.111,E2 44.1719} C_DIS
LIN {X 33.2985,Y 37.5828,Z 65,A 42.2468,B 24.8482,C -2.8426,E1 25.105,E2 41.2526} C_DIS
LIN {X 31.9867,Y 38.7053,Z 65,A 44.5862,B 24.847,C -2.8533,E1 25.1,E2 38.8967} C_DIS
LIN {X 29.1267,Y 40.9007,Z 65,A 48.8858,B 24.8459,C -2.8639,E1 25.0903,E2 34.5874} C_DIS
LIN {X 26.1075,Y 42.8909,Z 65,A 52.5017,B 24.8463,C -2.8605,E1 25.0818,E2 30.9912} C_DIS
LIN {X 24.1231,Y 44.038,Z 65,A 55.3333,B 24.8454,C -2.8681,E1 25.0749,E2 28.1499} C_DIS
LIN {X 21.5505,Y 45.3522,Z 65,A 58.5113,B 24.8452,C -2.8699,E1 25.0669,E2 24.9761} C_DIS
LIN {X 19.3544,Y 46.3321,Z 65,A 61.4411,B 24.8446,C -2.8763,E1 25.0594,E2 22.0383} C_DIS
LIN {X 15.9767,Y 47.6023,Z 65,A 64.95,B 24.8454,C -2.8689,E1 25.0503,E2 18.5542} C_DIS
LIN {X 13.5354,Y 48.3534,Z 65,A 68.5604,B 24.8438,C -2.8834,E1 25.0405,E2 14.9156} C_DIS
LIN {X 10.755,Y 49.0465,Z 65,A 71.9739,B 24.8433,C -2.8876,E1 25.0312,E2 11.4967} C_DIS
LIN {X 7.3332,Y 49.6742,Z 65,A 75.5867,B 24.8439,C -2.8826,E1 25.0213,E2 7.8996} C_DIS
LIN {X 5.411,Y 49.9198,Z 65,A 78.1222,B 24.8432,C -2.8886,E1 25.0142,E2 5.3515} C_DIS
LIN {X 1.2484,Y 50.1972,Z 65,A 82.0996,B 24.8447,C -2.8749,E1 25.0032,E2 1.408} C_DIS
LIN {X -1.9739,Y 50.1734,Z 65,A 86.2215,B 24.844,C -2.8816,E1 24.9917,E2 -2.73} C_DIS
LIN {X -4.667,Y 49.9945,Z 65,A 89.2803,B 24.8442,C -2.8798,E1 24.9832,E2 -5.786} C_DIS
LIN {X -7.4981,Y 49.6492,Z 65,A 92.5328,B 24.8444,C -2.8778,E1 24.9742,E2 -9.0362} C_DIS
LIN {X -9.5221,Y 49.3007,Z 65,A 94.5212,B 24.8452,C -2.8702,E1 24.9688,E2 -11.0085} C_DIS
LIN {X -11.8723,Y 48.7881,Z 65,A 97.9138,B 24.8443,C -2.8783,E1 24.9595,E2 -14.4249} C_DIS
LIN {X -14.8275,Y 47.9727,Z 65,A 101.7596,B 24.8441,C -2.8802,E1 24.9492,E2 -18.2816} C_DIS
LIN {X -19.3147,Y 46.3488,Z 65,A 106.3041,B 24.8465,C -2.8587,E1 24.9374,E2 -22.7844} C_DIS
LIN {X -20.7323,Y 45.732,Z 65,A 108.3945,B 24.8462,C -2.8612,E1 24.9321,E2 -24.886} C_DIS
LIN {X -23.5648,Y 44.3392,Z 65,A 111.5862,B 24.8475,C -2.8491,E1 24.9241,E2 -28.0573} C_DIS
LIN {X -25.5976,Y 43.1972,Z 65,A 115.0233,B 24.8467,C -2.8565,E1 24.9158,E2 -31.5223} C_DIS
LIN {X -28.6096,Y 41.2641,Z 65,A 118.6378,B 24.8483,C -2.8415,E1 24.9074,E2 -35.1129} C_DIS
LIN {X -30.3874,Y 39.9721,Z 65,A 121.2579,B 24.8487,C -2.8381,E1 24.9016,E2 -37.7343} C_DIS
LIN {X -32.5286,Y 38.2508,Z 65,A 124.2788,B 24.8496,C -2.8297,E1 24.8951,E2 -40.7465} C_DIS
LIN {X -34.1649,Y 36.796,Z 65,A 126.9862,B 24.8498,C -2.8272,E1 24.8895,E2 -43.4588} C_DIS
LIN {X -36.2177,Y 34.7781,Z 65,A 130.2239,B 24.8508,C -2.8187,E1 24.8831,E2 -46.6899} C_DIS
LIN {X -38.0222,Y 32.7952,Z 65,A 133.2247,B 24.8516,C -2.8102,E1 24.8776,E2 -49.684} C_DIS
LIN {X -39.5653,Y 30.9175,Z 65,A 136.3485,B 24.8519,C -2.8082,E1 24.8721,E2 -52.8176} C_DIS
LIN {X -41.6707,Y 28.0137,Z 65,A 140.5142,B 24.8529,C -2.7983,E1 24.8655,E2 -56.9801} C_DIS
LIN {X -42.9328,Y 26.0386,Z 65,A 143.2057,B 24.8537,C -2.7911,E1 24.8616,E2 -59.6682} C_DIS
LIN {X -44.837,Y 22.6041,Z 65,A 147.042,B 24.856,C -2.769,E1 24.8565,E2 -63.4719} C_DIS
LIN {X -45.7159,Y 20.7681,Z 65,A 149.6849,B 24.8562,C -2.7667,E1 24.8534,E2 -66.1239} C_DIS
LIN {X -46.6726,Y 18.5183,Z 65,A 152.5642,B 24.857,C -2.7597,E1 24.8503,E2 -69.0024} C_DIS
LIN {X -47.4614,Y 16.3922,Z 65,A 155.0142,B 24.858,C -2.7499,E1 24.848,E2 -71.4429} C_DIS
LIN {X -48.1537,Y 14.2288,Z 65,A 157.8056,B 24.8585,C -2.7448,E1 24.8458,E2 -74.2381} C_DIS
LIN {X -48.7974,Y 11.8344,Z 65,A 160.689,B 24.8593,C -2.7368,E1 24.8438,E2 -77.1193} C_DIS
LIN {X -49.4393,Y 8.7749,Z 65,A 164.7749,B 24.8597,C -2.7331,E1 24.8416,E2 -81.2204} C_DIS
LIN {X -49.9408,Y 5.2102,Z 65,A 168.3286,B 24.8618,C -2.7123,E1 24.8404,E2 -84.7456} C_DIS
LIN {X -50.1229,Y 2.9953,Z 65,A 171.4384,B 24.8618,C -2.7124,E1 24.8399,E2 -87.8745} C_DIS
LIN {X -50.1929,Y -1.388,Z 65,A 176.2178,B 24.8638,C -2.6936,E1 24.8399,E2 -92.6375} C_DIS
LIN {X -50.0182,Y -4.4079,Z 65,A 179.2851,B 24.8654,C -2.6773,E1 24.8406,E2 -95.6845} C_DIS
LIN {X -49.7632,Y -6.6994,Z 65,A -178.1697,B 24.8663,C -2.668,E1 24.8414,E2 -98.2225} C_DIS
LIN {X -49.504,Y -8.4021,Z 65,A -175.9375,B 24.8666,C -2.6658,E1 24.8424,E2 -100.4627} C_DIS
LIN {X -48.9944,Y -10.9927,Z 65,A -173.0036,B 24.8676,C -2.6555,E1 24.8441,E2 -103.3893} C_DIS
LIN {X -48.3531,Y -13.5362,Z 65,A -169.774,B 24.8681,C -2.65,E1 24.8464,E2 -106.6245} C_DIS
LIN {X -47.5768,Y -16.0525,Z 65,A -167.2127,B 24.8696,C -2.6348,E1 24.8486,E2 -109.1642} C_DIS
LIN {X -46.732,Y -18.3671,Z 65,A -163.5961,B 24.8693,C -2.6384,E1 24.8522,E2 -112.8098} C_DIS
LIN {X -45.3065,Y -21.6464,Z 65,A -160.2367,B 24.8714,C -2.6166,E1 24.856,E2 -116.1354} C_DIS
LIN {X -43.9733,Y -24.2415,Z 65,A -156.1375,B 24.8712,C -2.619,E1 24.8615,E2 -120.2622} C_DIS
LIN {X -42.1227,Y -27.33,Z 65,A -152.3048,B 24.8726,C -2.6044,E1 24.8671,E2 -124.0796} C_DIS
LIN {X -40.985,Y -29.0086,Z 65,A -149.9267,B 24.8731,C -2.5997,E1 24.8709,E2 -126.4581} C_DIS
LIN {X -39.3201,Y -31.2278,Z 65,A -146.8177,B 24.8739,C -2.5915,E1 24.8762,E2 -129.562} C_DIS
LIN {X -37.536,Y -33.3514,Z 65,A -143.8028,B 24.8748,C -2.5821,E1 24.8817,E2 -132.5683} C_DIS
LIN {X -35.061,Y -35.9436,Z 65,A -139.7364,B 24.8757,C -2.5732,E1 24.8897,E2 -136.6309} C_DIS
LIN {X -32.619,Y -38.1736,Z 65,A -136.0613,B 24.8765,C -2.5644,E1 24.8973,E2 -140.2995} C_DIS
LIN {X -30.7272,Y -39.7124,Z 65,A -133.0306,B 24.8766,C -2.5633,E1 24.9039,E2 -143.3389} C_DIS
LIN {X -28.6257,Y -41.2529,Z 65,A -129.7119,B 24.8766,C -2.5639,E1 24.9115,E2 -146.6706} C_DIS
LIN {X -25.3779,Y -43.327,Z 65,A -125.4797,B 24.8775,C -2.5549,E1 24.9216,E2 -150.8944} C_DIS
LIN {X -23.3223,Y -44.467,Z 65,A -122.9421,B 24.878,C -2.5491,E1 24.9278,E2 -153.4253} C_DIS
LIN {X -20.5984,Y -45.7923,Z 65,A -119.0066,B 24.8776,C -2.5531,E1 24.9378,E2 -157.3802} C_DIS
LIN {X -16.5607,Y -47.4023,Z 65,A -114.2894,B 24.8784,C -2.5446,E1 24.9501,E2 -162.0869} C_DIS
LIN {X -13.6434,Y -48.3228,Z 65,A -110.9007,B 24.8788,C -2.5405,E1 24.9592,E2 -165.4715} C_DIS
LIN {X -10.8983,Y -49.0153,Z 65,A -107.7477,B 24.8791,C -2.5375,E1 24.9678,E2 -168.6217} C_DIS
LIN {X -7.9238,Y -49.5834,Z 65,A -103.0604,B 24.8772,C -2.558,E1 24.9808,E2 -173.3621} C_DIS
LIN {X -4.2976,Y -50.0285,Z 65,A -99.419,B 24.8781,C -2.5484,E1 24.9909,E2 -176.9824} C_DIS
LIN {X -0.2559,Y -50.2112,Z 65,A -95.5867,B 24.8794,C -2.5351,E1 25.0015,E2 -180.7837} C_DIS
LIN {X -0.2559,Y -50.2112,Z 65,A -95.5867,B 24.8794,C -2.5351,E1 25.0015,E2 -180.7837} C_DIS
Enddeposition()
LIN {X 0.2375,Y -49.266,Z 65,A -95.3779,B 24.8784,C -2.5453,E1 25.0021,E2 -181.0164} C_DIS
Startdeposition()
$VEL.CP = VEL_PRINT
LIN {X -1.3067,Y -49.2525,Z 65,A -99.0309,B 24.8814,C -2.5134,E1 24.9917,E2 -177.2874} C_DIS
LIN {X -6.4241,Y -48.8489,Z 65,A -104.9923,B 24.8814,C -2.5142,E1 24.9752,E2 -171.3244} C_DIS
LIN {X -10.3833,Y -48.163,Z 65,A -109.2852,B 24.8806,C -2.5221,E1 24.9635,E2 -167.0456} C_DIS
LIN {X -13.9764,Y -47.2455,Z 65,A -112.5527,B 24.8787,C -2.5416,E1 24.9548,E2 -163.8195} C_DIS
LIN {X -16.1121,Y -46.5609,Z 65,A -116.1497,B 24.8801,C -2.5278,E1 24.9451,E2 -160.1829} C_DIS
LIN {X -18.7549,Y -45.5605,Z 65,A -119.2368,B 24.8795,C -2.534,E1 24.9371,E2 -157.104} C_DIS
LIN {X -21.3755,Y -44.391,Z 65,A -122.6277,B 24.8792,C -2.5369,E1 24.9285,E2 -153.7115} C_DIS
LIN {X -23.193,Y -43.4699,Z 65,A -125.1067,B 24.8791,C -2.5382,E1 24.9224,E2 -151.2288} C_DIS
LIN {X -26.7694,Y -41.3631,Z 65,A -129.736,B 24.8781,C -2.5482,E1 24.9114,E2 -146.609} C_DIS
LIN {X -29.403,Y -39.5343,Z 65,A -133.6703,B 24.8778,C -2.5513,E1 24.9024,E2 -142.6684} C_DIS
LIN {X -31.5179,Y -37.8695,Z 65,A -136.9384,B 24.8775,C -2.555,E1 24.8954,E2 -139.3966} C_DIS
LIN {X -33.8081,Y -35.8398,Z 65,A -141.2125,B 24.8778,C -2.5517,E1 24.8866,E2 -135.0972} C_DIS
LIN {X -36.416,Y -33.187,Z 65,A -144.4948,B 24.8754,C -2.5759,E1 24.8804,E2 -131.8583} C_DIS
LIN {X -38.4463,Y -30.8127,Z 65,A -149.041,B 24.8759,C -2.5712,E1 24.8723,E2 -127.2799} C_DIS
LIN {X -40.5768,Y -27.9471,Z 65,A -152.3375,B 24.8737,C -2.5933,E1 24.867,E2 -124.0201} C_DIS
LIN {X -41.9227,Y -25.8834,Z 65,A -155.5671,B 24.8735,C -2.5955,E1 24.8622,E2 -120.7794} C_DIS
LIN {X -44.2857,Y -21.5947,Z 65,A -160.5468,B 24.871,C -2.6207,E1 24.8557,E2 -115.8334} C_DIS
LIN {X -45.7553,Y -18.2736,Z 65,A -165.2798,B 24.8706,C -2.6255,E1 24.8504,E2 -111.0857} C_DIS
LIN {X -46.6283,Y -15.9156,Z 65,A -168.4149,B 24.87,C -2.631,E1 24.8475,E2 -107.9461} C_DIS
LIN {X -47.4521,Y -13.2591,Z 65,A -171.26,B 24.8685,C -2.6459,E1 24.8453,E2 -105.12} C_DIS
LIN {X -47.9523,Y -11.3171,Z 65,A -173.6354,B 24.8679,C -2.6523,E1 24.8437,E2 -102.7461} C_DIS
LIN {X -48.2917,Y -9.7673,Z 65,A -176.0365,B 24.8681,C -2.6504,E1 24.8424,E2 -100.3262} C_DIS
LIN {X -48.7522,Y -7.123,Z 65,A -178.7508,B 24.8666,C -2.6654,E1 24.8412,E2 -97.6318} C_DIS
LIN {X -49.1135,Y -3.9166,Z 65,A 176.9035,B 24.8662,C -2.6692,E1 24.84,E2 -93.269} C_DIS
LIN {X -49.2691,Y -0.0755,Z 65,A 173.0417,B 24.864,C -2.6913,E1 24.8398,E2 -89.4368} C_DIS
LIN {X -49.2133,Y 2.3438,Z 65,A 169.8416,B 24.8636,C -2.695,E1 24.8401,E2 -86.2263} C_DIS
LIN {X -48.959,Y 5.5253,Z 65,A 166.1648,B 24.8624,C -2.7071,E1 24.8411,E2 -82.5564} C_DIS
LIN {X -48.5132,Y 8.6001,Z 65,A 162.8136,B 24.8609,C -2.7219,E1 24.8426,E2 -79.2207} C_DIS
LIN {X -48.0252,Y 11.0015,Z 65,A 160.1278,B 24.8597,C -2.733,E1 24.8441,E2 -76.5456} C_DIS
LIN {X -47.6021,Y 12.7097,Z 65,A 157.4355,B 24.86,C -2.7307,E1 24.8461,E2 -73.8321} C_DIS
LIN {X -46.3541,Y 16.6974,Z 65,A 152.5287,B 24.8585,C -2.7448,E1 24.8504,E2 -68.9311} C_DIS
LIN {X -45.0849,Y 19.8702,Z 65,A 148.5465,B 24.8573,C -2.7565,E1 24.8547,E2 -64.9548} C_DIS
LIN {X -43.114,Y 23.8473,Z 65,A 143.2475,B 24.8559,C -2.7695,E1 24.8616,E2 -59.6586} C_DIS
LIN {X -41.6558,Y 26.3122,Z 65,A 139.6062,B 24.8554,C -2.7745,E1 24.867,E2 -56.0108} C_DIS
LIN {X -38.8823,Y 30.2605,Z 65,A 134.4793,B 24.8531,C -2.796,E1 24.8754,E2 -50.9105} C_DIS
LIN {X -36.5347,Y 33.0559,Z 65,A 130.8177,B 24.8512,C -2.8148,E1 24.882,E2 -47.2771} C_DIS
LIN {X -35.5385,Y 34.1247,Z 65,A 129.0083,B 24.8509,C -2.8174,E1 24.8855,E2 -45.466} C_DIS
LIN {X -34.431,Y 35.2421,Z 65,A 126.5827,B 24.8513,C -2.8132,E1 24.8904,E2 -43.0204} C_DIS
LIN {X -31.8643,Y 37.5786,Z 65,A 122.4084,B 24.8506,C -2.8202,E1 24.8991,E2 -38.8464} C_DIS
LIN {X -28.3537,Y 40.2933,Z 65,A 117.8294,B 24.8486,C -2.8391,E1 24.9093,E2 -34.296} C_DIS
LIN {X -25.5377,Y 42.1343,Z 65,A 113.0864,B 24.8491,C -2.8342,E1 24.9206,E2 -29.5264} C_DIS
LIN {X -21.8206,Y 44.1738,Z 65,A 108.9696,B 24.8469,C -2.8543,E1 24.9306,E2 -25.446} C_DIS
LIN {X -19.7816,Y 45.1239,Z 65,A 106.1685,B 24.8469,C -2.8554,E1 24.9378,E2 -22.6406} C_DIS
LIN {X -17.4931,Y 46.0594,Z 65,A 103.3028,B 24.8464,C -2.8593,E1 24.9452,E2 -19.7782} C_DIS
LIN {X -15.3048,Y 46.8322,Z 65,A 100.5919,B 24.8461,C -2.8624,E1 24.9524,E2 -17.0693} C_DIS
LIN {X -13.2996,Y 47.4406,Z 65,A 97.6476,B 24.8466,C -2.8571,E1 24.9603,E2 -14.1078} C_DIS
LIN {X -10.0048,Y 48.243,Z 65,A 94.662,B 24.8446,C -2.8756,E1 24.9683,E2 -11.1623} C_DIS
LIN {X -7.7245,Y 48.6605,Z 65,A 91.1089,B 24.8459,C -2.864,E1 24.9782,E2 -7.5781} C_DIS
LIN {X -4.6421,Y 49.0503,Z 65,A 87.7991,B 24.8452,C -2.8707,E1 24.9874,E2 -4.2824} C_DIS
LIN {X -1.0481,Y 49.2584,Z 65,A 83.2901,B 24.8456,C -2.8669,E1 25,E2 0.2367} C_DIS
LIN {X 3.6786,Y 49.1325,Z 65,A 77.3031,B 24.8464,C -2.8592,E1 25.0167,E2 6.24} C_DIS
LIN {X 8.9068,Y 48.4572,Z 65,A 71.6589,B 24.8457,C -2.8656,E1 25.0322,E2 11.8637} C_DIS
LIN {X 13.0745,Y 47.5032,Z 65,A 66.7354,B 24.8459,C -2.8636,E1 25.0455,E2 16.7847} C_DIS
LIN {X 15.7256,Y 46.6924,Z 65,A 63.6789,B 24.8459,C -2.8639,E1 25.0536,E2 19.8345} C_DIS
LIN {X 18.6256,Y 45.6132,Z 65,A 59.9496,B 24.8465,C -2.8582,E1 25.0634,E2 23.5693} C_DIS
LIN {X 22.1307,Y 44.0193,Z 65,A 55.9452,B 24.8462,C -2.8614,E1 25.0734,E2 27.5557} C_DIS
LIN {X 23.9195,Y 43.0737,Z 65,A 53.6717,B 24.8464,C -2.8597,E1 25.079,E2 29.8268} C_DIS
LIN {X 25.4158,Y 42.2084,Z 65,A 51.3965,B 24.8472,C -2.852,E1 25.0845,E2 32.1131} C_DIS
LIN {X 27.7446,Y 40.7148,Z 65,A 48.461,B 24.8472,C -2.8521,E1 25.0913,E2 35.0387} C_DIS
LIN {X 29.5647,Y 39.4132,Z 65,A 45.1073,B 24.8491,C -2.834,E1 25.0989,E2 38.4234} C_DIS
LIN {X 32.189,Y 37.3011,Z 65,A 41.1219,B 24.85,C -2.8254,E1 25.1074,E2 42.4137} C_DIS
LIN {X 34.9549,Y 34.7224,Z 65,A 36.9452,B 24.8506,C -2.8205,E1 25.1158,E2 46.5847} C_DIS
LIN {X 37.2605,Y 32.2363,Z 65,A 33.2942,B 24.8509,C -2.8172,E1 25.1226,E2 50.2271} C_DIS
LIN {X 38.7535,Y 30.4247,Z 65,A 30.9031,B 24.8509,C -2.8173,E1 25.1267,E2 52.6068} C_DIS
LIN {X 40.2335,Y 28.4386,Z 65,A 27.8039,B 24.8521,C -2.8062,E1 25.1318,E2 55.7175} C_DIS
LIN {X 41.5306,Y 26.5084,Z 65,A 25.3173,B 24.8524,C -2.8035,E1 25.1356,E2 58.1979} C_DIS
LIN {X 42.5253,Y 24.8819,Z 65,A 23.1839,B 24.8528,C -2.7994,E1 25.1387,E2 60.3301} C_DIS
LIN {X 43.662,Y 22.8281,Z 65,A 19.8856,B 24.8547,C -2.7811,E1 25.1431,E2 63.6544} C_DIS
LIN {X 45.3902,Y 19.1626,Z 65,A 15.1783,B 24.8561,C -2.7681,E1 25.1484,E2 68.3668} C_DIS
LIN {X 46.3099,Y 16.8187,Z 65,A 12.3567,B 24.8567,C -2.7618,E1 25.1512,E2 71.1877} C_DIS
LIN {X 47.4042,Y 13.4279,Z 65,A 9.2019,B 24.856,C -2.7691,E1 25.1538,E2 74.3073} C_DIS
LIN {X 47.9922,Y 11.1456,Z 65,A 5.513,B 24.8588,C -2.7421,E1 25.1563,E2 78.0386} C_DIS
LIN {X 48.4834,Y 8.7653,Z 65,A 2.9642,B 24.8591,C -2.739,E1 25.1576,E2 80.58} C_DIS
LIN {X 49.001,Y 5.1354,Z 65,A -1.6798,B 24.8612,C -2.7183,E1 25.1592,E2 85.2456} C_DIS
LIN {X 49.2691,Y 0.2208,Z 65,A -6.4565,B 24.8612,C -2.7192,E1 25.1598,E2 89.9917} C_DIS
LIN {X 49.2433,Y -1.6041,Z 65,A -9.0651,B 24.8628,C -2.7028,E1 25.1596,E2 92.6236} C_DIS
LIN {X 49.113,Y -3.9224,Z 65,A -11.4165,B 24.863,C -2.7012,E1 25.1592,E2 94.9646} C_DIS
LIN {X 48.7135,Y -7.3818,Z 65,A -15.4222,B 24.8642,C -2.6894,E1 25.1578,E2 98.9748} C_DIS
LIN {X 48.4799,Y -8.7849,Z 65,A -18.1517,B 24.8668,C -2.6629,E1 25.1564,E2 101.7509} C_DIS
LIN {X 47.5858,Y -12.7698,Z 65,A -22.5779,B 24.8677,C -2.6545,E1 25.1534,E2 106.1714} C_DIS
LIN {X 46.4024,Y -16.5594,Z 65,A -26.8264,B 24.8684,C -2.6477,E1 25.1497,E2 110.412} C_DIS
LIN {X 44.7484,Y -20.6173,Z 65,A -32.3013,B 24.8706,C -2.6251,E1 25.1436,E2 115.9104} C_DIS
LIN {X 43.2369,Y -23.6233,Z 65,A -35.5263,B 24.8704,C -2.6273,E1 25.1395,E2 119.1131} C_DIS
LIN {X 41.8728,Y -25.9648,Z 65,A -38.8618,B 24.8716,C -2.6148,E1 25.1346,E2 122.4611} C_DIS
LIN {X 39.8959,Y -28.9093,Z 65,A -43.4664,B 24.8736,C -2.5944,E1 25.1272,E2 127.0915} C_DIS
LIN {X 38.0623,Y -31.2859,Z 65,A -47.078,B 24.8747,C -2.583,E1 25.1209,E2 130.7133} C_DIS
LIN {X 34.7573,Y -34.9205,Z 65,A -51.4985,B 24.8737,C -2.5939,E1 25.1125,E2 135.0888} C_DIS
LIN {X 32.7672,Y -36.794,Z 65,A -55.8739,B 24.8766,C -2.5638,E1 25.1034,E2 139.5177} C_DIS
LIN {X 30.3028,Y -38.8497,Z 65,A -59.5531,B 24.8773,C -2.5568,E1 25.0953,E2 143.1998} C_DIS
LIN {X 26.569,Y -41.4917,Z 65,A -64.2744,B 24.8773,C -2.5576,E1 25.0845,E2 147.9033} C_DIS
LIN {X 23.9231,Y -43.0717,Z 65,A -67.6602,B 24.8775,C -2.5549,E1 25.0763,E2 151.2852} C_DIS
LIN {X 22.0024,Y -44.0838,Z 65,A -70.8429,B 24.879,C -2.5387,E1 25.0683,E2 154.4976} C_DIS
LIN {X 17.4933,Y -46.0593,Z 65,A -76.0728,B 24.879,C -2.5396,E1 25.0548,E2 159.7132} C_DIS
LIN {X 15.3125,Y -46.8288,Z 65,A -78.8766,B 24.8794,C -2.5343,E1 25.0474,E2 162.5242} C_DIS
LIN {X 11.7631,Y -47.8446,Z 65,A -82.8909,B 24.8794,C -2.5348,E1 25.0366,E2 166.5309} C_DIS
LIN {X 8.7613,Y -48.4842,Z 65,A -86.5819,B 24.8799,C -2.5296,E1 25.0265,E2 170.2297} C_DIS
LIN {X 6.0044,Y -48.9025,Z 65,A -90.659,B 24.8814,C -2.5132,E1 25.0151,E2 174.3425} C_DIS
LIN {X 2.4994,Y -49.2064,Z 65,A -93.8043,B 24.8801,C -2.5275,E1 25.0064,E2 177.4523} C_DIS
LIN {X 0.2375,Y -49.266,Z 65,A -95.3773,B 24.8784,C -2.545,E1 25.0022,E2 178.9835} C_DIS
Enddeposition()
LIN {X 0.2375,Y -49.266,Z 65,A -95.3773,B 24.8784,C -2.545,E1 25.0022,E2 178.9835} C_DIS
Startdeposition()
$VEL.CP = VEL_PRINT
LIN {X 1.5995,Y -48.3006,Z 65,A -93.4435,B 24.8763,C -2.5671,E1 25.0077,E2 176.9976} C_DIS
LIN {X 4.9239,Y -48.075,Z 65,A -89.5911,B 24.8763,C -2.5673,E1 25.0184,E2 173.1466} C_DIS
LIN {X 7.1214,Y -47.8001,Z 65,A -86.7253,B 24.8757,C -2.5733,E1 25.0264,E2 170.2693} C_DIS
LIN {X 10.1703,Y -47.2448,Z 65,A -83.2718,B 24.8757,C -2.5724,E1 25.0358,E2 166.8218} C_DIS
LIN {X 11.9854,Y -46.8169,Z 65,A -80.3649,B 24.8743,C -2.5871,E1 25.0438,E2 163.8845} C_DIS
LIN {X 16.4138,Y -45.4544,Z 65,A -75.4488,B 24.8747,C -2.5832,E1 25.0567,E2 158.9871} C_DIS
LIN {X 19.6138,Y -44.1679,Z 65,A -71.0821,B 24.8737,C -2.5941,E1 25.068,E2 154.6047} C_DIS
LIN {X 22.6928,Y -42.6681,Z 65,A -67.1477,B 24.8732,C -2.5984,E1 25.0778,E2 150.671} C_DIS
LIN {X 25.0454,Y -41.3306,Z 65,A -64.3612,B 24.8734,C -2.5963,E1 25.0845,E2 147.898} C_DIS
LIN {X 27.3982,Y -39.8106,Z 65,A -60.5484,B 24.8719,C -2.612,E1 25.0934,E2 144.0608} C_DIS
LIN {X 29.4592,Y -38.3099,Z 65,A -57.8247,B 24.8719,C -2.6126,E1 25.0994,E2 141.3456} C_DIS
LIN {X 30.937,Y -37.1263,Z 65,A -55.1564,B 24.8706,C -2.6256,E1 25.1052,E2 138.6567} C_DIS
LIN {X 33.9042,Y -34.4383,Z 65,A -50.5842,B 24.8698,C -2.6332,E1 25.1145,E2 134.0852} C_DIS
LIN {X 36.6401,Y -31.5116,Z 65,A -46.3387,B 24.8696,C -2.6352,E1 25.1224,E2 129.8538} C_DIS
LIN {X 37.8383,Y -30.0627,Z 65,A -44.2791,B 24.8694,C -2.6377,E1 25.126,E2 127.7979} C_DIS
LIN {X 39.3693,Y -28.0277,Z 65,A -40.6901,B 24.8675,C -2.6569,E1 25.132,E2 124.1808} C_DIS
LIN {X 40.9323,Y -25.6914,Z 65,A -37.8184,B 24.8675,C -2.6569,E1 25.1363,E2 121.3232} C_DIS
LIN {X 42.2923,Y -23.3852,Z 65,A -34.3732,B 24.866,C -2.6713,E1 25.1411,E2 117.8618} C_DIS
LIN {X 43.8364,Y -20.3436,Z 65,A -30.0173,B 24.8642,C -2.6894,E1 25.1464,E2 113.4867} C_DIS
LIN {X 45.1495,Y -17.2345,Z 65,A -25.9083,B 24.8627,C -2.7035,E1 25.1507,E2 109.3669} C_DIS
LIN {X 46.6503,Y -12.6188,Z 65,A -20.8252,B 24.8623,C -2.7078,E1 25.1548,E2 104.3028} C_DIS
LIN {X 47.3087,Y -9.8691,Z 65,A -17.3262,B 24.8609,C -2.7211,E1 25.1569,E2 100.7925} C_DIS
LIN {X 47.7331,Y -7.5547,Z 65,A -14.582,B 24.8601,C -2.729,E1 25.1582,E2 98.0459} C_DIS
LIN {X 48.144,Y -4.2067,Z 65,A -10.8088,B 24.8593,C -2.737,E1 25.1593,E2 94.2759} C_DIS
LIN {X 48.296,Y -1.7476,Z 65,A -8.0082,B 24.8586,C -2.7438,E1 25.1597,E2 91.4759} C_DIS
LIN {X 48.316,Y 1.0371,Z 65,A -4.262,B 24.8566,C -2.7631,E1 25.1597,E2 87.7064} C_DIS
LIN {X 48.0225,Y 5.4195,Z 65,A 1.5725,B 24.8536,C -2.7918,E1 25.1581,E2 81.8385} C_DIS
LIN {X 47.1111,Y 10.7722,Z 65,A 7.5147,B 24.8526,C -2.8015,E1 25.1549,E2 75.9082} C_DIS
LIN {X 46.0229,Y 14.7445,Z 65,A 12.1936,B 24.8515,C -2.8118,E1 25.1512,E2 71.2316} C_DIS
LIN {X 45.0245,Y 17.5582,Z 65,A 15.4423,B 24.851,C -2.8162,E1 25.148,E2 67.9905} C_DIS
LIN {X 43.9559,Y 20.085,Z 65,A 18.5098,B 24.8504,C -2.8217,E1 25.1446,E2 64.9268} C_DIS
LIN {X 42.8664,Y 22.3162,Z 65,A 21.5729,B 24.8493,C -2.832,E1 25.1408,E2 61.8556} C_DIS
LIN {X 41.7012,Y 24.4239,Z 65,A 24.3456,B 24.8487,C -2.8379,E1 25.1369,E2 59.0832} C_DIS
LIN {X 40.3361,Y 26.6175,Z 65,A 27.3071,B 24.8481,C -2.8437,E1 25.1325,E2 56.1228} C_DIS
LIN {X 39.1274,Y 28.3642,Z 65,A 30.0645,B 24.8469,C -2.8545,E1 25.128,E2 53.3535} C_DIS
LIN {X 37.9123,Y 29.9692,Z 65,A 32.6443,B 24.8459,C -2.8638,E1 25.1235,E2 50.7638} C_DIS
LIN {X 36.2542,Y 31.9557,Z 65,A 35.0054,B 24.8466,C -2.8573,E1 25.1193,E2 48.4288} C_DIS
LIN {X 34.0868,Y 34.258,Z 65,A 38.9414,B 24.8454,C -2.8687,E1 25.1116,E2 44.4826} C_DIS
LIN {X 32.2214,Y 36.0176,Z 65,A 42.2396,B 24.8442,C -2.8796,E1 25.1048,E2 41.1721} C_DIS
LIN {X 30.6845,Y 37.3366,Z 65,A 44.397,B 24.8442,C -2.8795,E1 25.1002,E2 39.0232} C_DIS
LIN {X 28.5582,Y 38.9862,Z 65,A 47.4398,B 24.8439,C -2.8824,E1 25.0935,E2 35.9846} C_DIS
LIN {X 26.3301,Y 40.5245,Z 65,A 51.2368,B 24.8422,C -2.8981,E1 25.0846,E2 32.1629} C_DIS
LIN {X 23.7156,Y 42.1081,Z 65,A 54.5362,B 24.8422,C -2.8974,E1 25.0767,E2 28.8754} C_DIS
LIN {X 21.4216,Y 43.3198,Z 65,A 57.2377,B 24.8426,C -2.8946,E1 25.07,E2 26.1879} C_DIS
LIN {X 19.9925,Y 43.9979,Z 65,A 59.3177,B 24.8419,C -2.9003,E1 25.0647,E2 24.0996} C_DIS
LIN {X 17.8949,Y 44.8923,Z 65,A 62.0154,B 24.8417,C -2.903,E1 25.0577,E2 21.4018} C_DIS
LIN {X 15.9655,Y 45.6135,Z 65,A 64.4006,B 24.8415,C -2.9041,E1 25.0515,E2 19.0188} C_DIS
LIN {X 14.1189,Y 46.2189,Z 65,A 66.9757,B 24.8408,C -2.9106,E1 25.0446,E2 16.4331} C_DIS
LIN {X 11.2623,Y 46.9966,Z 65,A 70.3457,B 24.8408,C -2.9102,E1 25.0355,E2 13.069} C_DIS
LIN {X 8.8963,Y 47.5016,Z 65,A 73.2423,B 24.8407,C -2.9119,E1 25.0276,E2 10.1719} C_DIS
LIN {X 6.3413,Y 47.9092,Z 65,A 75.9782,B 24.8412,C -2.9072,E1 25.0201,E2 7.4498} C_DIS
LIN {X 4.0872,Y 48.1542,Z 65,A 79.1156,B 24.8403,C -2.915,E1 25.0113,E2 4.2958} C_DIS
LIN {X 0.5803,Y 48.3243,Z 65,A 82.7585,B 24.8413,C -2.9061,E1 25.0012,E2 0.675} C_DIS
LIN {X -2.0923,Y 48.2816,Z 65,A 86.9806,B 24.8395,C -2.9223,E1 24.9893,E2 -3.5864} C_DIS
LIN {X -5.6137,Y 47.9998,Z 65,A 90.6787,B 24.8406,C -2.9123,E1 24.9791,E2 -7.2627} C_DIS
LIN {X -8.4539,Y 47.5815,Z 65,A 93.9787,B 24.8411,C -2.9083,E1 24.97,E2 -10.5561} C_DIS
LIN {X -11.1461,Y 47.0248,Z 65,A 97.2812,B 24.8413,C -2.9061,E1 24.961,E2 -13.8576} C_DIS
LIN {X -13.221,Y 46.4833,Z 65,A 99.42,B 24.8423,C -2.8973,E1 24.9553,E2 -15.9787} C_DIS
LIN {X -15.7476,Y 45.6886,Z 65,A 103.5111,B 24.8411,C -2.9082,E1 24.9444,E2 -20.1035} C_DIS
LIN {X -19.7491,Y 44.1075,Z 65,A 108.1746,B 24.8426,C -2.8944,E1 24.9324,E2 -24.7447} C_DIS
LIN {X -22.7449,Y 42.6406,Z 65,A 112.4387,B 24.8428,C -2.8927,E1 24.9218,E2 -29.0163} C_DIS
LIN {X -26.1488,Y 40.6415,Z 65,A 116.6603,B 24.8444,C -2.8775,E1 24.9118,E2 -33.2147} C_DIS
LIN {X -27.76,Y 39.558,Z 65,A 119.6497,B 24.8438,C -2.8831,E1 24.9049,E2 -36.2276} C_DIS
LIN {X -31.2,Y 36.9064,Z 65,A 124.7093,B 24.8452,C -2.8708,E1 24.894,E2 -41.2768} C_DIS
LIN {X -34.7073,Y 33.629,Z 65,A 129.3168,B 24.8482,C -2.8422,E1 24.8848,E2 -45.8351} C_DIS
LIN {X -36.7742,Y 31.3549,Z 65,A 134.1226,B 24.8475,C -2.8495,E1 24.8758,E2 -50.6799} C_DIS
LIN {X -39.2435,Y 28.2026,Z 65,A 138.77,B 24.8489,C -2.8356,E1 24.8681,E2 -55.3164} C_DIS
LIN {X -41.0933,Y 25.4336,Z 65,A 142.4081,B 24.8506,C -2.8204,E1 24.8626,E2 -58.9367} C_DIS
LIN {X -42.4766,Y 23.0476,Z 65,A 145.4541,B 24.8519,C -2.8081,E1 24.8584,E2 -61.9692} C_DIS
LIN {X -43.6195,Y 20.8051,Z 65,A 148.3258,B 24.8529,C -2.7979,E1 24.8549,E2 -64.8319} C_DIS
LIN {X -44.6064,Y 18.5949,Z 65,A 152.0587,B 24.8526,C -2.8012,E1 24.8508,E2 -68.5932} C_DIS
LIN {X -45.659,Y 15.8358,Z 65,A 155.3583,B 24.854,C -2.7878,E1 24.8477,E2 -71.8796} C_DIS
LIN {X -46.6761,Y 12.5235,Z 65,A 159.1065,B 24.8558,C -2.7703,E1 24.8448,E2 -75.6077} C_DIS
LIN {X -47.2467,Y 10.1618,Z 65,A 161.8585,B 24.857,C -2.7597,E1 24.8431,E2 -78.3503} C_DIS
LIN {X -47.589,Y 8.4142,Z 65,A 164.3879,B 24.857,C -2.7587,E1 24.8418,E2 -80.8924} C_DIS
LIN {X -48.0585,Y 5.0858,Z 65,A 168.2002,B 24.8586,C -2.7438,E1 24.8405,E2 -84.6919} C_DIS
LIN {X -48.3119,Y 1.2195,Z 65,A 173.5276,B 24.8591,C -2.7393,E1 24.8398,E2 -90.0405} C_DIS
LIN {X -48.2884,Y -1.9341,Z 65,A 176.3077,B 24.8616,C -2.7146,E1 24.84,E2 -92.7784} C_DIS
LIN {X -48.1716,Y -3.8712,Z 65,A 178.8557,B 24.862,C -2.7108,E1 24.8405,E2 -95.3325} C_DIS
LIN {X -47.9583,Y -5.9601,Z 65,A -178.7053,B 24.8628,C -2.7024,E1 24.8412,E2 -97.7661} C_DIS
LIN {X -47.6662,Y -7.9638,Z 65,A -175.742,B 24.8628,C -2.7027,E1 24.8426,E2 -100.7477} C_DIS
LIN {X -47.0084,Y -11.2125,Z 65,A -172.1475,B 24.8645,C -2.6862,E1 24.8447,E2 -104.3239} C_DIS
LIN {X -46.4063,Y -13.4912,Z 65,A -169.4017,B 24.8654,C -2.6773,E1 24.8468,E2 -107.0643} C_DIS
LIN {X -45.6791,Y -15.7785,Z 65,A -166.7853,B 24.8665,C -2.6659,E1 24.8491,E2 -109.6683} C_DIS
LIN {X -45.1717,Y -17.1758,Z 65,A -163.9359,B 24.8655,C -2.6759,E1 24.852,E2 -112.5577} C_DIS
LIN {X -43.5824,Y -20.8821,Z 65,A -159.6312,B 24.8675,C -2.656,E1 24.8569,E2 -116.8384} C_DIS
LIN {X -41.9306,Y -24.0274,Z 65,A -156.2396,B 24.8698,C -2.6333,E1 24.8614,E2 -120.1937} C_DIS
LIN {X -40.8088,Y -25.8882,Z 65,A -152.8715,B 24.8693,C -2.6378,E1 24.8664,E2 -123.5898} C_DIS
LIN {X -39.3148,Y -28.104,Z 65,A -149.3586,B 24.8696,C -2.6351,E1 24.872,E2 -127.1134} C_DIS
LIN {X -37.0733,Y -31.0013,Z 65,A -145.3839,B 24.8711,C -2.6197,E1 24.8789,E2 -131.0699} C_DIS
LIN {X -35.3752,Y -32.9264,Z 65,A -141.5582,B 24.8707,C -2.6246,E1 24.8863,E2 -134.9242} C_DIS
LIN {X -32.8324,Y -35.4622,Z 65,A -137.6742,B 24.872,C -2.6105,E1 24.8941,E2 -138.7905} C_DIS
LIN {X -30.6393,Y -37.3737,Z 65,A -135.034,B 24.8739,C -2.5921,E1 24.8997,E2 -141.3968} C_DIS
LIN {X -29.1028,Y -38.5814,Z 65,A -132.3931,B 24.8738,C -2.5929,E1 24.9055,E2 -144.0494} C_DIS
LIN {X -27.1999,Y -39.9458,Z 65,A -129.9091,B 24.8746,C -2.584,E1 24.9112,E2 -146.5206} C_DIS
LIN {X -23.9976,Y -41.9477,Z 65,A -125.0646,B 24.8747,C -2.5831,E1 24.9228,E2 -151.378} C_DIS
LIN {X -21.5778,Y -43.2423,Z 65,A -122.0679,B 24.8755,C -2.5751,E1 24.9302,E2 -154.3637} C_DIS
LIN {X -19.812,Y -44.0792,Z 65,A -119.79,B 24.8758,C -2.5719,E1 24.9359,E2 -156.6397} C_DIS
LIN {X -18.0257,Y -44.8397,Z 65,A -117.3824,B 24.8758,C -2.5713,E1 24.9422,E2 -159.0512} C_DIS
LIN {X -15.7241,Y -45.6978,Z 65,A -114.1378,B 24.8756,C -2.5741,E1 24.9507,E2 -162.3091} C_DIS
LIN {X -13.2667,Y -46.4703,Z 65,A -111.0817,B 24.8758,C -2.5721,E1 24.9589,E2 -165.3655} C_DIS
LIN {X -10.0436,Y -47.2724,Z 65,A -107.4852,B 24.8765,C -2.5646,E1 24.9686,E2 -168.9488} C_DIS
LIN {X -8.2879,Y -47.6117,Z 65,A -104.6939,B 24.8755,C -2.575,E1 24.9764,E2 -171.7676} C_DIS
LIN {X -3.7375,Y -48.1823,Z 65,A -99.6476,B 24.8762,C -2.5678,E1 24.9904,E2 -176.8} C_DIS
Enddeposition()
END
